LIN {X 0,Y 242.578,Z 857.441,A -85,B 0,C 180,E1 -19152.29,E2 -19152.29} C_VEL
LIN {X 0,Y 241.483,Z 861.061,A -85,B 0,C 180,E1 -19154.816,E2 -19154.816} C_VEL
LIN {X 0,Y 240.352,Z 864.916,A -85,B 0,C 180,E1 -19158.189,E2 -19158.189} C_VEL
LIN {X 0,Y 239.899,Z 867.777,A -85,B 0,C 180,E1 -19161.577,E2 -19161.577} C_VEL
LIN {X 0,Y 239.797,Z 869.672,A -85,B 0,C 180,E1 -19164.956,E2 -19164.956} C_VEL
LIN {X 0,Y 239.756,Z 870.35,A -85,B 0,C 180,E1 -19166.639,E2 -19166.639} C_VEL
LIN {X 0,Y 239.862,Z 870.828,A -85,B 0,C 180,E1 -19170,E2 -19170} C_VEL
LIN {X 0,Y 239.756,Z 870.35,A -85,B 0,C 180,E1 -19173.361,E2 -19173.361} C_VEL
LIN {X 0,Y 239.78,Z 868.917,A -85,B 0,C 180,E1 -19176.733,E2 -19176.733} C_VEL
LIN {X 0,Y 240.067,Z 866.522,A -85,B 0,C 180,E1 -19180.116,E2 -19180.116} C_VEL
LIN {X 0,Y 241.126,Z 862.101,A -85,B 0,C 180,E1 -19184.344,E2 -19184.344} C_VEL
LIN {X 0,Y 242.159,Z 858.729,A -85,B 0,C 180,E1 -19186.871,E2 -19186.871} C_VEL
LIN {X 0,Y 244.064,Z 853.224,A -85,B 0,C 180,E1 -19190.215,E2 -19190.215} C_VEL
LIN {X 0,Y 245.911,Z 848.361,A -85,B 0,C 180,E1 -19192.694,E2 -19192.694} C_VEL
LIN {X 0,Y 248.516,Z 841.742,A -85,B 0,C 180,E1 -19195.547,E2 -19195.547} C_VEL
LIN {X 0,Y 251.72,Z 834.036,A -85,B 0,C 180,E1 -19198.335,E2 -19198.335} C_VEL
LIN {X 0,Y 254.947,Z 826.486,A -85,B 0,C 180,E1 -19200.662,E2 -19200.662} C_VEL
LIN {X 0,Y 258.438,Z 817.9,A -85,B 0,C 180,E1 -19202.947,E2 -19202.947} C_VEL
LIN {X 0,Y 262.348,Z 808.111,A -85,B 0,C 180,E1 -19205.166,E2 -19205.166} C_VEL
LIN {X 0,Y 266.73,Z 796.887,A -85,B 0,C 180,E1 -19207.301,E2 -19207.301} C_VEL
LIN {X 0,Y 270.235,Z 787.33,A -85,B 0,C 180,E1 -19208.859,E2 -19208.859} C_VEL
LIN {X 0,Y 273.955,Z 776.523,A -85,B 0,C 180,E1 -19210.372,E2 -19210.372} C_VEL
LIN {X 0,Y 277.393,Z 765.586,A -85,B 0,C 180,E1 -19211.686,E2 -19211.686} C_VEL
LIN {X 0,Y 281.007,Z 752.933,A -85,B 0,C 180,E1 -19212.962,E2 -19212.962} C_VEL
LIN {X 0,Y 283.803,Z 741.946,A -85,B 0,C 180,E1 -19213.897,E2 -19213.897} C_VEL
LIN {X 0,Y 286.488,Z 729.861,A -85,B 0,C 180,E1 -19214.76,E2 -19214.76} C_VEL
LIN {X 0,Y 289.158,Z 715.743,A -85,B 0,C 180,E1 -19215.557,E2 -19215.557} C_VEL
LIN {X 0,Y 291.186,Z 702.376,A -85,B 0,C 180,E1 -19216.14,E2 -19216.14} C_VEL
LIN {X 0,Y 292.661,Z 688.923,A -85,B 0,C 180,E1 -19216.586,E2 -19216.586} C_VEL
LIN {X 0,Y 295.022,Z 651.638,A -85,B 0,C 180,E1 -19217.474,E2 -19217.474} C_VEL
LIN {X 0,Y 299.994,Z 567.021,A -85,B 0,C 180,E1 -19219.406,E2 -19219.406} C_VEL
LIN {X 0,Y 293.621,Z 552.933,A -85,B 0,C 180,E1 -19221.404,E2 -19221.404} C_VEL
LIN {X 0,Y 286.94,Z 539.628,A -85,B 0,C 180,E1 -19223.638,E2 -19223.638} C_VEL
LIN {X 0,Y 280.747,Z 528.524,A -85,B 0,C 180,E1 -19225.868,E2 -19225.868} C_VEL
LIN {X 0,Y 275.075,Z 519.016,A -85,B 0,C 180,E1 -19228.092,E2 -19228.092} C_VEL
LIN {X 0,Y 271.322,Z 513.261,A -85,B 0,C 180,E1 -19229.67,E2 -19229.67} C_VEL
LIN {X 0,Y 268.084,Z 508.973,A -85,B 0,C 180,E1 -19231.095,E2 -19231.095} C_VEL
LIN {X 0,Y 264.624,Z 504.496,A -85,B 0,C 180,E1 -19232.727,E2 -19232.727} C_VEL
LIN {X 0,Y 261.902,Z 501.009,A -85,B 0,C 180,E1 -19234.107,E2 -19234.107} C_VEL
LIN {X 0,Y 260.988,Z 499.86,A -85,B 0,C 180,E1 -19234.591,E2 -19234.591} C_VEL
LIN {X 0,Y 258.194,Z 496.863,A -85,B 0,C 180,E1 -19236.115,E2 -19236.115} C_VEL
LIN {X 0,Y 256.919,Z 494.86,A -85,B 0,C 180,E1 -19236.898,E2 -19236.898} C_VEL
LIN {X 0,Y 254.24,Z 492.546,A -85,B 0,C 180,E1 -19238.514,E2 -19238.514} C_VEL
LIN {X 0,Y 252.29,Z 489.301,A -85,B 0,C 180,E1 -19239.915,E2 -19239.915} C_VEL
LIN {X 0,Y 249.327,Z 487.104,A -85,B 0,C 180,E1 -19242.043,E2 -19242.043} C_VEL
LIN {X 0,Y 247.221,Z 483.628,A -85,B 0,C 180,E1 -19243.944,E2 -19243.944} C_VEL
LIN {X 0,Y 244.135,Z 481.605,A -85,B 0,C 180,E1 -19246.897,E2 -19246.897} C_VEL
LIN {X 0,Y 242.709,Z 479.452,A -85,B 0,C 180,E1 -19248.728,E2 -19248.728} C_VEL
LIN {X 0,Y 242.346,Z 478.039,A -85,B 0,C 180,E1 -19249.979,E2 -19249.979} C_VEL
LIN {X 0,Y 242.395,Z 477.56,A -85,B 0,C 180,E1 -19251.664,E2 -19251.664} C_VEL
LIN {X 0,Y 242.252,Z 477.542,A -85,B 0,C 180,E1 -19255.007,E2 -19255.007} C_VEL
LIN {X 0,Y 242.631,Z 477.502,A -85,B 0,C 180,E1 -19258.34,E2 -19258.34} C_VEL
LIN {X 0,Y 242.631,Z 477.483,A -85,B 0,C 180,E1 -19261.659,E2 -19261.659} C_VEL
LIN {X 0,Y 242.423,Z 477.508,A -85,B 0,C 180,E1 -19266.703,E2 -19266.703} C_VEL
LIN {X 0,Y 242.362,Z 477.788,A -85,B 0,C 180,E1 -19270.019,E2 -19270.019} C_VEL
LIN {X 0,Y 242.547,Z 478.94,A -85,B 0,C 180,E1 -19271.384,E2 -19271.384} C_VEL
LIN {X 0,Y 243.957,Z 481.47,A -85,B 0,C 180,E1 -19273.324,E2 -19273.324} C_VEL
LIN {X 0,Y 247.548,Z 484.008,A -85,B 0,C 180,E1 -19276.767,E2 -19276.767} C_VEL
LIN {X 0,Y 249.333,Z 487.146,A -85,B 0,C 180,E1 -19278.381,E2 -19278.381} C_VEL
LIN {X 0,Y 251.923,Z 489.174,A -85,B 0,C 180,E1 -19280.264,E2 -19280.264} C_VEL
LIN {X 0,Y 252.55,Z 489.767,A -85,B 0,C 180,E1 -19280.697,E2 -19280.697} C_VEL
LIN {X 0,Y 254.388,Z 492.805,A -85,B 0,C 180,E1 -19282.005,E2 -19282.005} C_VEL
LIN {X 0,Y 257.319,Z 495.333,A -85,B 0,C 180,E1 -19283.756,E2 -19283.756} C_VEL
LIN {X 0,Y 259.737,Z 498.727,A -85,B 0,C 180,E1 -19285.17,E2 -19285.17} C_VEL
LIN {X 0,Y 261.606,Z 500.6,A -85,B 0,C 180,E1 -19286.151,E2 -19286.151} C_VEL
LIN {X 0,Y 264.594,Z 504.494,A -85,B 0,C 180,E1 -19287.676,E2 -19287.676} C_VEL
LIN {X 0,Y 266.072,Z 506.379,A -85,B 0,C 180,E1 -19288.388,E2 -19288.388} C_VEL
LIN {X 0,Y 269.712,Z 511.008,A -85,B 0,C 180,E1 -19290.043,E2 -19290.043} C_VEL
LIN {X 0,Y 273.86,Z 516.542,A -85,B 0,C 180,E1 -19291.795,E2 -19291.795} C_VEL
LIN {X 0,Y 284.021,Z 529.623,A -85,B 0,C 180,E1 -19295.55,E2 -19295.55} C_VEL
LIN {X 0,Y 290.619,Z 536.586,A -85,B 0,C 180,E1 -19297.623,E2 -19297.623} C_VEL
LIN {X 0,Y 297.294,Z 542.946,A -85,B 0,C 180,E1 -19299.585,E2 -19299.585} C_VEL
LIN {X 0,Y 301.355,Z 546.585,A -85,B 0,C 180,E1 -19300.818,E2 -19300.818} C_VEL
LIN {X 0,Y 308.526,Z 553.049,A -85,B 0,C 180,E1 -19303.171,E2 -19303.171} C_VEL
LIN {X 0,Y 314.885,Z 558.94,A -85,B 0,C 180,E1 -19305.464,E2 -19305.464} C_VEL
LIN {X 0,Y 319.671,Z 563.42,A -85,B 0,C 180,E1 -19307.347,E2 -19307.347} C_VEL
LIN {X 0,Y 325.679,Z 569.287,A -85,B 0,C 180,E1 -19309.852,E2 -19309.852} C_VEL
LIN {X 0,Y 328.38,Z 571.697,A -85,B 0,C 180,E1 -19310.998,E2 -19310.998} C_VEL
LIN {X 0,Y 333.028,Z 576.13,A -85,B 0,C 180,E1 -19313.027,E2 -19313.027} C_VEL
LIN {X 0,Y 336.117,Z 578.85,A -85,B 0,C 180,E1 -19314.418,E2 -19314.418} C_VEL
LIN {X 0,Y 340.541,Z 582.947,A -85,B 0,C 180,E1 -19316.493,E2 -19316.493} C_VEL
LIN {X 0,Y 343.794,Z 585.63,A -85,B 0,C 180,E1 -19318.061,E2 -19318.061} C_VEL
LIN {X 0,Y 347.343,Z 589.012,A -85,B 0,C 180,E1 -19319.866,E2 -19319.866} C_VEL
LIN {X 0,Y 351.211,Z 592.136,A -85,B 0,C 180,E1 -19321.908,E2 -19321.908} C_VEL
LIN {X 0,Y 355.329,Z 596.17,A -85,B 0,C 180,E1 -19324.268,E2 -19324.268} C_VEL
LIN {X 0,Y 359.603,Z 599.246,A -85,B 0,C 180,E1 -19326.871,E2 -19326.871} C_VEL
LIN {X 0,Y 362.933,Z 602.606,A -85,B 0,C 180,E1 -19329.176,E2 -19329.176} C_VEL
LIN {X 0,Y 366.336,Z 605.042,A -85,B 0,C 180,E1 -19331.682,E2 -19331.682} C_VEL
LIN {X 0,Y 368.406,Z 606.343,A -85,B 0,C 180,E1 -19333.373,E2 -19333.373} C_VEL
LIN {X 0,Y 370.835,Z 609.08,A -85,B 0,C 180,E1 -19335.737,E2 -19335.737} C_VEL
LIN {X 0,Y 373.171,Z 611.039,A -85,B 0,C 180,E1 -19338.326,E2 -19338.326} C_VEL
LIN {X 0,Y 375.093,Z 612.069,A -85,B 0,C 180,E1 -19340.883,E2 -19340.883} C_VEL
LIN {X 0,Y 376.609,Z 612.81,A -85,B 0,C 180,E1 -19343.571,E2 -19343.571} C_VEL
LIN {X 0,Y 377.431,Z 613.376,A -85,B 0,C 180,E1 -19345.729,E2 -19345.729} C_VEL
LIN {X 0,Y 377.962,Z 613.558,A -85,B 0,C 180,E1 -19347.869,E2 -19347.869} C_VEL
LIN {X 0,Y 378.149,Z 613.625,A -85,B 0,C 180,E1 -19350,E2 -19350} C_VEL
LIN {X 0,Y 377.962,Z 613.559,A -85,B 0,C 180,E1 -19352.131,E2 -19352.131} C_VEL
LIN {X 0,Y 377.274,Z 613.269,A -85,B 0,C 180,E1 -19354.781,E2 -19354.781} C_VEL
LIN {X 0,Y 376.055,Z 612.562,A -85,B 0,C 180,E1 -19357.517,E2 -19357.517} C_VEL
LIN {X 0,Y 374.23,Z 611.679,A -85,B 0,C 180,E1 -19360.35,E2 -19360.35} C_VEL
LIN {X 0,Y 372.082,Z 610.203,A -85,B 0,C 180,E1 -19362.92,E2 -19362.92} C_VEL
LIN {X 0,Y 369.668,Z 607.864,A -85,B 0,C 180,E1 -19365.436,E2 -19365.436} C_VEL
LIN {X 0,Y 367.787,Z 605.761,A -85,B 0,C 180,E1 -19367.17,E2 -19367.17} C_VEL
LIN {X 0,Y 364.975,Z 604.141,A -85,B 0,C 180,E1 -19369.345,E2 -19369.345} C_VEL
LIN {X 0,Y 361.445,Z 601.277,A -85,B 0,C 180,E1 -19371.867,E2 -19371.867} C_VEL
LIN {X 0,Y 358.801,Z 598.546,A -85,B 0,C 180,E1 -19373.638,E2 -19373.638} C_VEL
LIN {X 0,Y 354.828,Z 595.742,A -85,B 0,C 180,E1 -19376.017,E2 -19376.017} C_VEL
LIN {X 0,Y 350.884,Z 591.778,A -85,B 0,C 180,E1 -19378.28,E2 -19378.28} C_VEL
LIN {X 0,Y 345.972,Z 587.873,A -85,B 0,C 180,E1 -19380.832,E2 -19380.832} C_VEL
LIN {X 0,Y 342.068,Z 584.093,A -85,B 0,C 180,E1 -19382.788,E2 -19382.788} C_VEL
LIN {X 0,Y 337.417,Z 580.192,A -85,B 0,C 180,E1 -19384.975,E2 -19384.975} C_VEL
LIN {X 0,Y 333.911,Z 576.796,A -85,B 0,C 180,E1 -19386.585,E2 -19386.585} C_VEL
LIN {X 0,Y 328.966,Z 572.338,A -85,B 0,C 180,E1 -19388.746,E2 -19388.746} C_VEL
LIN {X 0,Y 326.272,Z 569.703,A -85,B 0,C 180,E1 -19389.911,E2 -19389.911} C_VEL
LIN {X 0,Y 321.823,Z 565.579,A -85,B 0,C 180,E1 -19391.758,E2 -19391.758} C_VEL
LIN {X 0,Y 318.346,Z 562.26,A -85,B 0,C 180,E1 -19393.185,E2 -19393.185} C_VEL
LIN {X 0,Y 312.159,Z 556.385,A -85,B 0,C 180,E1 -19395.543,E2 -19395.543} C_VEL
LIN {X 0,Y 307.422,Z 551.98,A -85,B 0,C 180,E1 -19397.201,E2 -19397.201} C_VEL
LIN {X 0,Y 300.789,Z 546.044,A -85,B 0,C 180,E1 -19399.361,E2 -19399.361} C_VEL
LIN {X 0,Y 293.324,Z 539.281,A -85,B 0,C 180,E1 -19401.584,E2 -19401.584} C_VEL
LIN {X 0,Y 285.505,Z 531.293,A -85,B 0,C 180,E1 -19403.962,E2 -19403.962} C_VEL
LIN {X 0,Y 279.921,Z 524.607,A -85,B 0,C 180,E1 -19405.877,E2 -19405.877} C_VEL
LIN {X 0,Y 271.593,Z 513.467,A -85,B 0,C 180,E1 -19409.148,E2 -19409.148} C_VEL
LIN {X 0,Y 268.299,Z 509.207,A -85,B 0,C 180,E1 -19410.584,E2 -19410.584} C_VEL
LIN {X 0,Y 264.715,Z 504.61,A -85,B 0,C 180,E1 -19412.267,E2 -19412.267} C_VEL
LIN {X 0,Y 261.77,Z 500.861,A -85,B 0,C 180,E1 -19413.759,E2 -19413.759} C_VEL
LIN {X 0,Y 260.849,Z 499.688,A -85,B 0,C 180,E1 -19414.25,E2 -19414.25} C_VEL
LIN {X 0,Y 258.122,Z 496.718,A -85,B 0,C 180,E1 -19415.745,E2 -19415.745} C_VEL
LIN {X 0,Y 256.853,Z 494.821,A -85,B 0,C 180,E1 -19416.519,E2 -19416.519} C_VEL
LIN {X 0,Y 254.103,Z 492.457,A -85,B 0,C 180,E1 -19418.183,E2 -19418.183} C_VEL
LIN {X 0,Y 252.405,Z 489.438,A -85,B 0,C 180,E1 -19419.418,E2 -19419.418} C_VEL
LIN {X 0,Y 249.7,Z 487.548,A -85,B 0,C 180,E1 -19421.328,E2 -19421.328} C_VEL
LIN {X 0,Y 247.993,Z 484.981,A -85,B 0,C 180,E1 -19422.795,E2 -19422.795} C_VEL
LIN {X 0,Y 247.164,Z 483.61,A -85,B 0,C 180,E1 -19423.575,E2 -19423.575} C_VEL
LIN {X 0,Y 243.957,Z 481.47,A -85,B 0,C 180,E1 -19426.676,E2 -19426.676} C_VEL
LIN {X 0,Y 242.598,Z 479.136,A -85,B 0,C 180,E1 -19428.512,E2 -19428.512} C_VEL
LIN {X 0,Y 242.338,Z 478.057,A -85,B 0,C 180,E1 -19429.558,E2 -19429.558} C_VEL
LIN {X 0,Y 242.381,Z 477.587,A -85,B 0,C 180,E1 -19430.764,E2 -19430.764} C_VEL
LIN {X 0,Y 242.426,Z 477.509,A -85,B 0,C 180,E1 -19433.341,E2 -19433.341} C_VEL
LIN {X 0,Y 242.631,Z 477.485,A -85,B 0,C 180,E1 -19438.341,E2 -19438.341} C_VEL
LIN {X 0,Y 242.631,Z 477.504,A -85,B 0,C 180,E1 -19441.66,E2 -19441.66} C_VEL
LIN {X 0,Y 242.419,Z 477.527,A -85,B 0,C 180,E1 -19446.66,E2 -19446.66} C_VEL
LIN {X 0,Y 242.373,Z 477.818,A -85,B 0,C 180,E1 -19449.645,E2 -19449.645} C_VEL
LIN {X 0,Y 242.593,Z 479.137,A -85,B 0,C 180,E1 -19451.066,E2 -19451.066} C_VEL
LIN {X 0,Y 244.132,Z 481.628,A -85,B 0,C 180,E1 -19453.103,E2 -19453.103} C_VEL
LIN {X 0,Y 247.528,Z 483.951,A -85,B 0,C 180,E1 -19456.33,E2 -19456.33} C_VEL
LIN {X 0,Y 249.449,Z 487.231,A -85,B 0,C 180,E1 -19458.054,E2 -19458.054} C_VEL
LIN {X 0,Y 252.537,Z 489.602,A -85,B 0,C 180,E1 -19460.26,E2 -19460.26} C_VEL
LIN {X 0,Y 254.346,Z 492.684,A -85,B 0,C 180,E1 -19461.556,E2 -19461.556} C_VEL
LIN {X 0,Y 257.375,Z 495.471,A -85,B 0,C 180,E1 -19463.378,E2 -19463.378} C_VEL
LIN {X 0,Y 259.718,Z 498.74,A -85,B 0,C 180,E1 -19464.747,E2 -19464.747} C_VEL
LIN {X 0,Y 261.594,Z 500.527,A -85,B 0,C 180,E1 -19465.725,E2 -19465.725} C_VEL
LIN {X 0,Y 264.253,Z 504.142,A -85,B 0,C 180,E1 -19467.097,E2 -19467.097} C_VEL
LIN {X 0,Y 265.821,Z 505.972,A -85,B 0,C 180,E1 -19467.848,E2 -19467.848} C_VEL
LIN {X 0,Y 269.791,Z 511.206,A -85,B 0,C 180,E1 -19469.666,E2 -19469.666} C_VEL
LIN {X 0,Y 273.093,Z 515.902,A -85,B 0,C 180,E1 -19471.085,E2 -19471.085} C_VEL
LIN {X 0,Y 278.448,Z 524.496,A -85,B 0,C 180,E1 -19473.249,E2 -19473.249} C_VEL
LIN {X 0,Y 285.75,Z 537.328,A -85,B 0,C 180,E1 -19475.943,E2 -19475.943} C_VEL
LIN {X 0,Y 292.568,Z 550.783,A -85,B 0,C 180,E1 -19478.256,E2 -19478.256} C_VEL
LIN {X 0,Y 298.601,Z 563.806,A -85,B 0,C 180,E1 -19480.166,E2 -19480.166} C_VEL
LIN {X 0,Y 300.007,Z 567.051,A -85,B 0,C 180,E1 -19480.598,E2 -19480.598} C_VEL
LIN {X 0,Y 299.387,Z 577.69,A -85,B 0,C 180,E1 -19480.842,E2 -19480.842} C_VEL
LIN {X 0,Y 298.645,Z 583.54,A -85,B 0,C 180,E1 -19480.889,E2 -19480.889} C_VEL
LIN {X 0,Y 293.745,Z 602.654,A -85,B 0,C 180,E1 -19480.488,E2 -19480.488} C_VEL
LIN {X 0,Y 292.942,Z 608.51,A -85,B 0,C 180,E1 -19480.521,E2 -19480.521} C_VEL
LIN {X 0,Y 288.087,Z 685.999,A -85,B 0,C 180,E1 -19482.314,E2 -19482.314} C_VEL
LIN {X 0,Y 286.556,Z 700.167,A -85,B 0,C 180,E1 -19482.759,E2 -19482.759} C_VEL
LIN {X 0,Y 284.599,Z 713.234,A -85,B 0,C 180,E1 -19483.306,E2 -19483.306} C_VEL
LIN {X 0,Y 282.221,Z 725.93,A -85,B 0,C 180,E1 -19483.989,E2 -19483.989} C_VEL
LIN {X 0,Y 279.53,Z 738.313,A -85,B 0,C 180,E1 -19484.83,E2 -19484.83} C_VEL
LIN {X 0,Y 276.776,Z 749.24,A -85,B 0,C 180,E1 -19485.711,E2 -19485.711} C_VEL
LIN {X 0,Y 273.496,Z 760.877,A -85,B 0,C 180,E1 -19486.83,E2 -19486.83} C_VEL
LIN {X 0,Y 269.896,Z 772.398,A -85,B 0,C 180,E1 -19488.145,E2 -19488.145} C_VEL
LIN {X 0,Y 265.937,Z 783.688,A -85,B 0,C 180,E1 -19489.65,E2 -19489.65} C_VEL
LIN {X 0,Y 261.659,Z 795.329,A -85,B 0,C 180,E1 -19491.519,E2 -19491.519} C_VEL
LIN {X 0,Y 257.983,Z 804.349,A -85,B 0,C 180,E1 -19493.179,E2 -19493.179} C_VEL
LIN {X 0,Y 253.717,Z 814.554,A -85,B 0,C 180,E1 -19495.4,E2 -19495.4} C_VEL
LIN {X 0,Y 249.883,Z 823.512,A -85,B 0,C 180,E1 -19497.699,E2 -19497.699} C_VEL
LIN {X 0,Y 246.478,Z 831.405,A -85,B 0,C 180,E1 -19500.068,E2 -19500.068} C_VEL
LIN {X 0,Y 243.37,Z 838.369,A -85,B 0,C 180,E1 -19502.482,E2 -19502.482} C_VEL
LIN {X 0,Y 240.696,Z 844.59,A -85,B 0,C 180,E1 -19504.992,E2 -19504.992} C_VEL
LIN {X 0,Y 237.885,Z 851.464,A -85,B 0,C 180,E1 -19508.328,E2 -19508.328} C_VEL
LIN {X 0,Y 235.709,Z 857.228,A -85,B 0,C 180,E1 -19511.756,E2 -19511.756} C_VEL
LIN {X 0,Y 234.186,Z 861.889,A -85,B 0,C 180,E1 -19515.222,E2 -19515.222} C_VEL
LIN {X 0,Y 233.017,Z 866.311,A -85,B 0,C 180,E1 -19519.574,E2 -19519.574} C_VEL
LIN {X 0,Y 232.698,Z 868.707,A -85,B 0,C 180,E1 -19523.061,E2 -19523.061} C_VEL
LIN {X 0,Y 232.666,Z 870.14,A -85,B 0,C 180,E1 -19526.537,E2 -19526.537} C_VEL
LIN {X 0,Y 232.774,Z 870.619,A -85,B 0,C 180,E1 -19530,E2 -19530} C_VEL
LIN {X 0,Y 232.665,Z 870.14,A -85,B 0,C 180,E1 -19533.463,E2 -19533.463} C_VEL
LIN {X 0,Y 232.698,Z 868.706,A -85,B 0,C 180,E1 -19536.939,E2 -19536.939} C_VEL
LIN {X 0,Y 233.014,Z 866.311,A -85,B 0,C 180,E1 -19540.426,E2 -19540.426} C_VEL
LIN {X 0,Y 234.166,Z 861.888,A -85,B 0,C 180,E1 -19544.78,E2 -19544.78} C_VEL
LIN {X 0,Y 235.706,Z 857.227,A -85,B 0,C 180,E1 -19548.244,E2 -19548.244} C_VEL
LIN {X 0,Y 237.901,Z 851.464,A -85,B 0,C 180,E1 -19551.67,E2 -19551.67} C_VEL
LIN {X 0,Y 240.979,Z 843.955,A -85,B 0,C 180,E1 -19555.298,E2 -19555.298} C_VEL
LIN {X 0,Y 244.858,Z 835.031,A -85,B 0,C 180,E1 -19558.735,E2 -19558.735} C_VEL
LIN {X 0,Y 248.754,Z 826.272,A -85,B 0,C 180,E1 -19561.511,E2 -19561.511} C_VEL
LIN {X 0,Y 252.424,Z 817.687,A -85,B 0,C 180,E1 -19563.837,E2 -19563.837} C_VEL
LIN {X 0,Y 256.496,Z 807.898,A -85,B 0,C 180,E1 -19566.092,E2 -19566.092} C_VEL
LIN {X 0,Y 260.665,Z 797.681,A -85,B 0,C 180,E1 -19568.078,E2 -19568.078} C_VEL
LIN {X 0,Y 264.707,Z 787.119,A -85,B 0,C 180,E1 -19569.83,E2 -19569.83} C_VEL
LIN {X 0,Y 268.551,Z 776.312,A -85,B 0,C 180,E1 -19571.359,E2 -19571.359} C_VEL
LIN {X 0,Y 272.086,Z 765.375,A -85,B 0,C 180,E1 -19572.689,E2 -19572.689} C_VEL
LIN {X 0,Y 275.833,Z 752.723,A -85,B 0,C 180,E1 -19573.971,E2 -19573.971} C_VEL
LIN {X 0,Y 279.014,Z 740.52,A -85,B 0,C 180,E1 -19575.002,E2 -19575.002} C_VEL
LIN {X 0,Y 281.833,Z 728.015,A -85,B 0,C 180,E1 -19575.876,E2 -19575.876} C_VEL
LIN {X 0,Y 284.361,Z 714.767,A -85,B 0,C 180,E1 -19576.615,E2 -19576.615} C_VEL
LIN {X 0,Y 286.316,Z 702.167,A -85,B 0,C 180,E1 -19577.164,E2 -19577.164} C_VEL
LIN {X 0,Y 287.821,Z 688.713,A -85,B 0,C 180,E1 -19577.614,E2 -19577.614} C_VEL
LIN {X 0,Y 290.268,Z 651.428,A -85,B 0,C 180,E1 -19578.508,E2 -19578.508} C_VEL
LIN {X 0,Y 295.232,Z 570.658,A -85,B 0,C 180,E1 -19580.353,E2 -19580.353} C_VEL
LIN {X 0,Y 295.075,Z 569.346,A -85,B 0,C 180,E1 -19580.439,E2 -19580.439} C_VEL
LIN {X 0,Y 289.66,Z 557.204,A -85,B 0,C 180,E1 -19582.22,E2 -19582.22} C_VEL
LIN {X 0,Y 283.403,Z 544.435,A -85,B 0,C 180,E1 -19584.409,E2 -19584.409} C_VEL
LIN {X 0,Y 277.395,Z 533.505,A -85,B 0,C 180,E1 -19586.666,E2 -19586.666} C_VEL
LIN {X 0,Y 272.283,Z 524.699,A -85,B 0,C 180,E1 -19588.758,E2 -19588.758} C_VEL
LIN {X 0,Y 268.629,Z 519.018,A -85,B 0,C 180,E1 -19590.354,E2 -19590.354} C_VEL
LIN {X 0,Y 265.723,Z 515.06,A -85,B 0,C 180,E1 -19591.684,E2 -19591.684} C_VEL
LIN {X 0,Y 262.691,Z 511.029,A -85,B 0,C 180,E1 -19593.162,E2 -19593.162} C_VEL
LIN {X 0,Y 259.678,Z 507.134,A -85,B 0,C 180,E1 -19594.739,E2 -19594.739} C_VEL
LIN {X 0,Y 255.903,Z 502.701,A -85,B 0,C 180,E1 -19596.881,E2 -19596.881} C_VEL
LIN {X 0,Y 255.059,Z 501.423,A -85,B 0,C 180,E1 -19597.416,E2 -19597.416} C_VEL
LIN {X 0,Y 252.353,Z 498.873,A -85,B 0,C 180,E1 -19599.122,E2 -19599.122} C_VEL
LIN {X 0,Y 250.721,Z 496.044,A -85,B 0,C 180,E1 -19600.344,E2 -19600.344} C_VEL
LIN {X 0,Y 247.866,Z 493.803,A -85,B 0,C 180,E1 -19602.466,E2 -19602.466} C_VEL
LIN {X 0,Y 245.972,Z 490.48,A -85,B 0,C 180,E1 -19604.244,E2 -19604.244} C_VEL
LIN {X 0,Y 243.004,Z 488.542,A -85,B 0,C 180,E1 -19607.154,E2 -19607.154} C_VEL
LIN {X 0,Y 241.462,Z 486.137,A -85,B 0,C 180,E1 -19609.2,E2 -19609.2} C_VEL
LIN {X 0,Y 240.567,Z 484.589,A -85,B 0,C 180,E1 -19610.625,E2 -19610.625} C_VEL
LIN {X 0,Y 237.598,Z 482.494,A -85,B 0,C 180,E1 -19618.305,E2 -19618.305} C_VEL
LIN {X 0,Y 237.552,Z 482.451,A -85,B 0,C 180,E1 -19621.695,E2 -19621.695} C_VEL
LIN {X 0,Y 240.611,Z 484.615,A -85,B 0,C 180,E1 -19629.858,E2 -19629.858} C_VEL
LIN {X 0,Y 241.398,Z 486.024,A -85,B 0,C 180,E1 -19631.12,E2 -19631.12} C_VEL
LIN {X 0,Y 243.095,Z 488.685,A -85,B 0,C 180,E1 -19633.372,E2 -19633.372} C_VEL
LIN {X 0,Y 246.11,Z 490.714,A -85,B 0,C 180,E1 -19636.308,E2 -19636.308} C_VEL
LIN {X 0,Y 247.758,Z 493.692,A -85,B 0,C 180,E1 -19637.861,E2 -19637.861} C_VEL
LIN {X 0,Y 250.398,Z 495.956,A -85,B 0,C 180,E1 -19639.859,E2 -19639.859} C_VEL
LIN {X 0,Y 251.045,Z 496.8,A -85,B 0,C 180,E1 -19640.338,E2 -19640.338} C_VEL
LIN {X 0,Y 253.246,Z 499.978,A -85,B 0,C 180,E1 -19641.895,E2 -19641.895} C_VEL
LIN {X 0,Y 255.524,Z 502.015,A -85,B 0,C 180,E1 -19643.289,E2 -19643.289} C_VEL
LIN {X 0,Y 258.351,Z 505.71,A -85,B 0,C 180,E1 -19644.96,E2 -19644.96} C_VEL
LIN {X 0,Y 259.726,Z 507.27,A -85,B 0,C 180,E1 -19645.708,E2 -19645.708} C_VEL
LIN {X 0,Y 262.821,Z 511.168,A -85,B 0,C 180,E1 -19647.318,E2 -19647.318} C_VEL
LIN {X 0,Y 267.62,Z 517.578,A -85,B 0,C 180,E1 -19649.606,E2 -19649.606} C_VEL
LIN {X 0,Y 270.907,Z 522.015,A -85,B 0,C 180,E1 -19651.043,E2 -19651.043} C_VEL
LIN {X 0,Y 281.495,Z 535.867,A -85,B 0,C 180,E1 -19655.092,E2 -19655.092} C_VEL
LIN {X 0,Y 287.919,Z 542.744,A -85,B 0,C 180,E1 -19657.166,E2 -19657.166} C_VEL
LIN {X 0,Y 295.192,Z 549.568,A -85,B 0,C 180,E1 -19659.295,E2 -19659.295} C_VEL
LIN {X 0,Y 302.425,Z 556.061,A -85,B 0,C 180,E1 -19661.525,E2 -19661.525} C_VEL
LIN {X 0,Y 305.86,Z 559.068,A -85,B 0,C 180,E1 -19662.644,E2 -19662.644} C_VEL
LIN {X 0,Y 310.698,Z 563.406,A -85,B 0,C 180,E1 -19664.317,E2 -19664.317} C_VEL
LIN {X 0,Y 316.854,Z 569.239,A -85,B 0,C 180,E1 -19666.633,E2 -19666.633} C_VEL
LIN {X 0,Y 319.938,Z 572.14,A -85,B 0,C 180,E1 -19667.879,E2 -19667.879} C_VEL
LIN {X 0,Y 324.807,Z 576.641,A -85,B 0,C 180,E1 -19669.898,E2 -19669.898} C_VEL
LIN {X 0,Y 331.048,Z 582.552,A -85,B 0,C 180,E1 -19672.593,E2 -19672.593} C_VEL
LIN {X 0,Y 334.327,Z 585.361,A -85,B 0,C 180,E1 -19674.047,E2 -19674.047} C_VEL
LIN {X 0,Y 338.74,Z 589.487,A -85,B 0,C 180,E1 -19676.087,E2 -19676.087} C_VEL
LIN {X 0,Y 342.282,Z 592.37,A -85,B 0,C 180,E1 -19677.779,E2 -19677.779} C_VEL
LIN {X 0,Y 345.934,Z 595.822,A -85,B 0,C 180,E1 -19679.627,E2 -19679.627} C_VEL
LIN {X 0,Y 349.861,Z 598.969,A -85,B 0,C 180,E1 -19681.672,E2 -19681.672} C_VEL
LIN {X 0,Y 353.995,Z 602.979,A -85,B 0,C 180,E1 -19684.034,E2 -19684.034} C_VEL
LIN {X 0,Y 358.415,Z 606.21,A -85,B 0,C 180,E1 -19686.701,E2 -19686.701} C_VEL
LIN {X 0,Y 361.742,Z 609.481,A -85,B 0,C 180,E1 -19688.965,E2 -19688.965} C_VEL
LIN {X 0,Y 365.198,Z 611.969,A -85,B 0,C 180,E1 -19691.481,E2 -19691.481} C_VEL
LIN {X 0,Y 367.292,Z 613.234,A -85,B 0,C 180,E1 -19693.172,E2 -19693.172} C_VEL
LIN {X 0,Y 369.659,Z 615.916,A -85,B 0,C 180,E1 -19695.443,E2 -19695.443} C_VEL
LIN {X 0,Y 372.051,Z 617.909,A -85,B 0,C 180,E1 -19698.008,E2 -19698.008} C_VEL
LIN {X 0,Y 374.024,Z 619.031,A -85,B 0,C 180,E1 -19700.607,E2 -19700.607} C_VEL
LIN {X 0,Y 375.395,Z 619.698,A -85,B 0,C 180,E1 -19702.855,E2 -19702.855} C_VEL
LIN {X 0,Y 376.404,Z 620.322,A -85,B 0,C 180,E1 -19705.208,E2 -19705.208} C_VEL
LIN {X 0,Y 377.097,Z 620.604,A -85,B 0,C 180,E1 -19707.864,E2 -19707.864} C_VEL
LIN {X 0,Y 377.284,Z 620.671,A -85,B 0,C 180,E1 -19710,E2 -19710} C_VEL
LIN {X 0,Y 377.097,Z 620.604,A -85,B 0,C 180,E1 -19712.136,E2 -19712.136} C_VEL
LIN {X 0,Y 376.404,Z 620.315,A -85,B 0,C 180,E1 -19714.793,E2 -19714.793} C_VEL
LIN {X 0,Y 375.174,Z 619.606,A -85,B 0,C 180,E1 -19717.535,E2 -19717.535} C_VEL
LIN {X 0,Y 373.344,Z 618.716,A -85,B 0,C 180,E1 -19720.375,E2 -19720.375} C_VEL
LIN {X 0,Y 371.178,Z 617.229,A -85,B 0,C 180,E1 -19722.952,E2 -19722.952} C_VEL
LIN {X 0,Y 368.74,Z 614.945,A -85,B 0,C 180,E1 -19725.476,E2 -19725.476} C_VEL
LIN {X 0,Y 366.978,Z 612.865,A -85,B 0,C 180,E1 -19727.109,E2 -19727.109} C_VEL
LIN {X 0,Y 364.011,Z 611.208,A -85,B 0,C 180,E1 -19729.396,E2 -19729.396} C_VEL
LIN {X 0,Y 360.329,Z 608.252,A -85,B 0,C 180,E1 -19732.005,E2 -19732.005} C_VEL
LIN {X 0,Y 357.56,Z 605.426,A -85,B 0,C 180,E1 -19733.848,E2 -19733.848} C_VEL
LIN {X 0,Y 353.634,Z 602.681,A -85,B 0,C 180,E1 -19736.174,E2 -19736.174} C_VEL
LIN {X 0,Y 349.592,Z 598.655,A -85,B 0,C 180,E1 -19738.48,E2 -19738.48} C_VEL
LIN {X 0,Y 344.431,Z 594.52,A -85,B 0,C 180,E1 -19741.147,E2 -19741.147} C_VEL
LIN {X 0,Y 340.545,Z 590.849,A -85,B 0,C 180,E1 -19743.056,E2 -19743.056} C_VEL
LIN {X 0,Y 335.681,Z 586.75,A -85,B 0,C 180,E1 -19745.332,E2 -19745.332} C_VEL
LIN {X 0,Y 332.197,Z 583.426,A -85,B 0,C 180,E1 -19746.914,E2 -19746.914} C_VEL
LIN {X 0,Y 327.107,Z 578.852,A -85,B 0,C 180,E1 -19749.121,E2 -19749.121} C_VEL
LIN {X 0,Y 324.594,Z 576.41,A -85,B 0,C 180,E1 -19750.192,E2 -19750.192} C_VEL
LIN {X 0,Y 320.057,Z 572.252,A -85,B 0,C 180,E1 -19752.072,E2 -19752.072} C_VEL
LIN {X 0,Y 316.857,Z 569.206,A -85,B 0,C 180,E1 -19753.368,E2 -19753.368} C_VEL
LIN {X 0,Y 311.828,Z 564.352,A -85,B 0,C 180,E1 -19755.287,E2 -19755.287} C_VEL
LIN {X 0,Y 306.361,Z 559.567,A -85,B 0,C 180,E1 -19757.184,E2 -19757.184} C_VEL
LIN {X 0,Y 302.676,Z 556.242,A -85,B 0,C 180,E1 -19758.397,E2 -19758.397} C_VEL
LIN {X 0,Y 297.62,Z 551.673,A -85,B 0,C 180,E1 -19759.97,E2 -19759.97} C_VEL
LIN {X 0,Y 290.602,Z 545.429,A -85,B 0,C 180,E1 -19762.03,E2 -19762.03} C_VEL
LIN {X 0,Y 282.646,Z 537.176,A -85,B 0,C 180,E1 -19764.518,E2 -19764.518} C_VEL
LIN {X 0,Y 277.149,Z 530.482,A -85,B 0,C 180,E1 -19766.466,E2 -19766.466} C_VEL
LIN {X 0,Y 269.11,Z 519.565,A -85,B 0,C 180,E1 -19769.732,E2 -19769.732} C_VEL
LIN {X 0,Y 265.849,Z 515.227,A -85,B 0,C 180,E1 -19771.209,E2 -19771.209} C_VEL
LIN {X 0,Y 262.353,Z 510.71,A -85,B 0,C 180,E1 -19772.91,E2 -19772.91} C_VEL
LIN {X 0,Y 258.77,Z 506.065,A -85,B 0,C 180,E1 -19774.817,E2 -19774.817} C_VEL
LIN {X 0,Y 255.96,Z 502.753,A -85,B 0,C 180,E1 -19776.432,E2 -19776.432} C_VEL
LIN {X 0,Y 254.918,Z 501.331,A -85,B 0,C 180,E1 -19777.082,E2 -19777.082} C_VEL
LIN {X 0,Y 252.128,Z 498.64,A -85,B 0,C 180,E1 -19778.857,E2 -19778.857} C_VEL
LIN {X 0,Y 250.629,Z 496.115,A -85,B 0,C 180,E1 -19779.98,E2 -19779.98} C_VEL
LIN {X 0,Y 247.872,Z 493.859,A -85,B 0,C 180,E1 -19782.041,E2 -19782.041} C_VEL
LIN {X 0,Y 246.151,Z 490.824,A -85,B 0,C 180,E1 -19783.648,E2 -19783.648} C_VEL
LIN {X 0,Y 242.499,Z 487.971,A -85,B 0,C 180,E1 -19787.34,E2 -19787.34} C_VEL
LIN {X 0,Y 240.749,Z 484.834,A -85,B 0,C 180,E1 -19789.913,E2 -19789.913} C_VEL
LIN {X 0,Y 238.882,Z 483.667,A -85,B 0,C 180,E1 -19793.242,E2 -19793.242} C_VEL
LIN {X 0,Y 237.554,Z 482.432,A -85,B 0,C 180,E1 -19798.305,E2 -19798.305} C_VEL
LIN {X 0,Y 237.644,Z 482.643,A -85,B 0,C 180,E1 -19802.119,E2 -19802.119} C_VEL
LIN {X 0,Y 240.562,Z 484.6,A -85,B 0,C 180,E1 -19809.37,E2 -19809.37} C_VEL
LIN {X 0,Y 241.46,Z 486.151,A -85,B 0,C 180,E1 -19810.8,E2 -19810.8} C_VEL
LIN {X 0,Y 243.091,Z 488.651,A -85,B 0,C 180,E1 -19812.948,E2 -19812.948} C_VEL
LIN {X 0,Y 246.219,Z 490.88,A -85,B 0,C 180,E1 -19815.997,E2 -19815.997} C_VEL
LIN {X 0,Y 247.867,Z 493.798,A -85,B 0,C 180,E1 -19817.534,E2 -19817.534} C_VEL
LIN {X 0,Y 250.909,Z 496.406,A -85,B 0,C 180,E1 -19819.805,E2 -19819.805} C_VEL
LIN {X 0,Y 253.09,Z 499.777,A -85,B 0,C 180,E1 -19821.375,E2 -19821.375} C_VEL
LIN {X 0,Y 255.505,Z 502.014,A -85,B 0,C 180,E1 -19822.863,E2 -19822.863} C_VEL
LIN {X 0,Y 258.255,Z 505.647,A -85,B 0,C 180,E1 -19824.494,E2 -19824.494} C_VEL
LIN {X 0,Y 259.759,Z 507.304,A -85,B 0,C 180,E1 -19825.31,E2 -19825.31} C_VEL
LIN {X 0,Y 262.873,Z 511.192,A -85,B 0,C 180,E1 -19826.926,E2 -19826.926} C_VEL
LIN {X 0,Y 267.586,Z 517.608,A -85,B 0,C 180,E1 -19829.179,E2 -19829.179} C_VEL
LIN {X 0,Y 270.501,Z 521.857,A -85,B 0,C 180,E1 -19830.474,E2 -19830.474} C_VEL
LIN {X 0,Y 275.882,Z 530.82,A -85,B 0,C 180,E1 -19832.731,E2 -19832.731} C_VEL
LIN {X 0,Y 282.246,Z 542.147,A -85,B 0,C 180,E1 -19835.166,E2 -19835.166} C_VEL
LIN {X 0,Y 289.088,Z 556.038,A -85,B 0,C 180,E1 -19837.588,E2 -19837.588} C_VEL
LIN {X 0,Y 294.539,Z 568.037,A -85,B 0,C 180,E1 -19839.387,E2 -19839.387} C_VEL
LIN {X 0,Y 295.202,Z 569.643,A -85,B 0,C 180,E1 -19839.602,E2 -19839.602} C_VEL
LIN {X 0,Y 292.942,Z 608.51,A -85,B 0,C 180,E1 -19840.521,E2 -19840.521} C_VEL
LIN {X 0,Y 292.136,Z 614.368,A -85,B 0,C 180,E1 -19840.553,E2 -19840.553} C_VEL
LIN {X 0,Y 287.172,Z 633.471,A -85,B 0,C 180,E1 -19840.119,E2 -19840.119} C_VEL
LIN {X 0,Y 286.372,Z 639.328,A -85,B 0,C 180,E1 -19840.153,E2 -19840.153} C_VEL
LIN {X 0,Y 283.213,Z 687.144,A -85,B 0,C 180,E1 -19841.287,E2 -19841.287} C_VEL
LIN {X 0,Y 281.653,Z 700.957,A -85,B 0,C 180,E1 -19841.736,E2 -19841.736} C_VEL
LIN {X 0,Y 279.637,Z 713.79,A -85,B 0,C 180,E1 -19842.284,E2 -19842.284} C_VEL
LIN {X 0,Y 277.285,Z 725.873,A -85,B 0,C 180,E1 -19842.939,E2 -19842.939} C_VEL
LIN {X 0,Y 274.599,Z 737.857,A -85,B 0,C 180,E1 -19843.753,E2 -19843.753} C_VEL
LIN {X 0,Y 271.698,Z 749.029,A -85,B 0,C 180,E1 -19844.657,E2 -19844.657} C_VEL
LIN {X 0,Y 268.313,Z 760.665,A -85,B 0,C 180,E1 -19845.783,E2 -19845.783} C_VEL
LIN {X 0,Y 264.149,Z 773.491,A -85,B 0,C 180,E1 -19847.278,E2 -19847.278} C_VEL
LIN {X 0,Y 260.084,Z 784.62,A -85,B 0,C 180,E1 -19848.803,E2 -19848.803} C_VEL
LIN {X 0,Y 256.458,Z 794.126,A -85,B 0,C 180,E1 -19850.339,E2 -19850.339} C_VEL
LIN {X 0,Y 252.256,Z 804.136,A -85,B 0,C 180,E1 -19852.199,E2 -19852.199} C_VEL
LIN {X 0,Y 247.838,Z 814.342,A -85,B 0,C 180,E1 -19854.457,E2 -19854.457} C_VEL
LIN {X 0,Y 243.81,Z 823.299,A -85,B 0,C 180,E1 -19856.792,E2 -19856.792} C_VEL
LIN {X 0,Y 240.253,Z 831.192,A -85,B 0,C 180,E1 -19859.209,E2 -19859.209} C_VEL
LIN {X 0,Y 236.994,Z 838.155,A -85,B 0,C 180,E1 -19861.675,E2 -19861.675} C_VEL
LIN {X 0,Y 234.249,Z 844.21,A -85,B 0,C 180,E1 -19864.167,E2 -19864.167} C_VEL
LIN {X 0,Y 231.207,Z 851.251,A -85,B 0,C 180,E1 -19867.669,E2 -19867.669} C_VEL
LIN {X 0,Y 228.878,Z 857.015,A -85,B 0,C 180,E1 -19871.191,E2 -19871.191} C_VEL
LIN {X 0,Y 227.627,Z 860.635,A -85,B 0,C 180,E1 -19873.867,E2 -19873.867} C_VEL
LIN {X 0,Y 226.331,Z 864.492,A -85,B 0,C 180,E1 -19877.446,E2 -19877.446} C_VEL
LIN {X 0,Y 225.752,Z 867.354,A -85,B 0,C 180,E1 -19881.045,E2 -19881.045} C_VEL
LIN {X 0,Y 225.587,Z 869.25,A -85,B 0,C 180,E1 -19884.637,E2 -19884.637} C_VEL
LIN {X 0,Y 225.58,Z 869.93,A -85,B 0,C 180,E1 -19886.428,E2 -19886.428} C_VEL
LIN {X 0,Y 225.688,Z 870.409,A -85,B 0,C 180,E1 -19890,E2 -19890} C_VEL
LIN {X 0,Y 225.579,Z 869.93,A -85,B 0,C 180,E1 -19893.572,E2 -19893.572} C_VEL
LIN {X 0,Y 225.607,Z 868.495,A -85,B 0,C 180,E1 -19897.158,E2 -19897.158} C_VEL
LIN {X 0,Y 225.979,Z 866.099,A -85,B 0,C 180,E1 -19900.754,E2 -19900.754} C_VEL
LIN {X 0,Y 227.23,Z 861.676,A -85,B 0,C 180,E1 -19905.242,E2 -19905.242} C_VEL
LIN {X 0,Y 228.396,Z 858.303,A -85,B 0,C 180,E1 -19907.921,E2 -19907.921} C_VEL
LIN {X 0,Y 230.545,Z 852.796,A -85,B 0,C 180,E1 -19911.457,E2 -19911.457} C_VEL
LIN {X 0,Y 232.642,Z 847.934,A -85,B 0,C 180,E1 -19914.068,E2 -19914.068} C_VEL
LIN {X 0,Y 236,Z 840.261,A -85,B 0,C 180,E1 -19917.489,E2 -19917.489} C_VEL
LIN {X 0,Y 239.116,Z 833.609,A -85,B 0,C 180,E1 -19919.977,E2 -19919.977} C_VEL
LIN {X 0,Y 242.626,Z 826.059,A -85,B 0,C 180,E1 -19922.403,E2 -19922.403} C_VEL
LIN {X 0,Y 246.445,Z 817.473,A -85,B 0,C 180,E1 -19924.774,E2 -19924.774} C_VEL
LIN {X 0,Y 250.734,Z 807.686,A -85,B 0,C 180,E1 -19927.058,E2 -19927.058} C_VEL
LIN {X 0,Y 255.053,Z 797.469,A -85,B 0,C 180,E1 -19929.073,E2 -19929.073} C_VEL
LIN {X 0,Y 259.235,Z 786.907,A -85,B 0,C 180,E1 -19930.846,E2 -19930.846} C_VEL
LIN {X 0,Y 263.195,Z 776.099,A -85,B 0,C 180,E1 -19932.394,E2 -19932.394} C_VEL
LIN {X 0,Y 266.879,Z 765.164,A -85,B 0,C 180,E1 -19933.729,E2 -19933.729} C_VEL
LIN {X 0,Y 270.247,Z 754.253,A -85,B 0,C 180,E1 -19934.861,E2 -19934.861} C_VEL
LIN {X 0,Y 273.714,Z 741.525,A -85,B 0,C 180,E1 -19935.966,E2 -19935.966} C_VEL
LIN {X 0,Y 276.623,Z 729.258,A -85,B 0,C 180,E1 -19936.843,E2 -19936.843} C_VEL
LIN {X 0,Y 279.388,Z 715.323,A -85,B 0,C 180,E1 -19937.639,E2 -19937.639} C_VEL
LIN {X 0,Y 281.541,Z 701.957,A -85,B 0,C 180,E1 -19938.223,E2 -19938.223} C_VEL
LIN {X 0,Y 283.088,Z 688.504,A -85,B 0,C 180,E1 -19938.675,E2 -19938.675} C_VEL
LIN {X 0,Y 285.618,Z 651.219,A -85,B 0,C 180,E1 -19939.574,E2 -19939.574} C_VEL
LIN {X 0,Y 290.593,Z 572.371,A -85,B 0,C 180,E1 -19941.396,E2 -19941.396} C_VEL
LIN {X 0,Y 284.57,Z 558.845,A -85,B 0,C 180,E1 -19943.484,E2 -19943.484} C_VEL
LIN {X 0,Y 278.81,Z 547.184,A -85,B 0,C 180,E1 -19945.617,E2 -19945.617} C_VEL
LIN {X 0,Y 272.143,Z 534.849,A -85,B 0,C 180,E1 -19948.307,E2 -19948.307} C_VEL
LIN {X 0,Y 266.427,Z 525.4,A -85,B 0,C 180,E1 -19950.844,E2 -19950.844} C_VEL
LIN {X 0,Y 263.105,Z 520.843,A -85,B 0,C 180,E1 -19952.417,E2 -19952.417} C_VEL
LIN {X 0,Y 260.082,Z 516.841,A -85,B 0,C 180,E1 -19953.953,E2 -19953.953} C_VEL
LIN {X 0,Y 256.954,Z 512.671,A -85,B 0,C 180,E1 -19955.677,E2 -19955.677} C_VEL
LIN {X 0,Y 254.016,Z 509.117,A -85,B 0,C 180,E1 -19957.425,E2 -19957.425} C_VEL
LIN {X 0,Y 253.14,Z 507.95,A -85,B 0,C 180,E1 -19957.988,E2 -19957.988} C_VEL
LIN {X 0,Y 250.31,Z 504.907,A -85,B 0,C 180,E1 -19959.876,E2 -19959.876} C_VEL
LIN {X 0,Y 249.06,Z 502.744,A -85,B 0,C 180,E1 -19960.85,E2 -19960.85} C_VEL
LIN {X 0,Y 246.195,Z 500.203,A -85,B 0,C 180,E1 -19963.093,E2 -19963.093} C_VEL
LIN {X 0,Y 244.677,Z 497.361,A -85,B 0,C 180,E1 -19964.589,E2 -19964.589} C_VEL
LIN {X 0,Y 241.879,Z 495.476,A -85,B 0,C 180,E1 -19967.413,E2 -19967.413} C_VEL
LIN {X 0,Y 240.305,Z 492.985,A -85,B 0,C 180,E1 -19969.574,E2 -19969.574} C_VEL
LIN {X 0,Y 239.557,Z 491.568,A -85,B 0,C 180,E1 -19970.826,E2 -19970.826} C_VEL
LIN {X 0,Y 236.733,Z 489.544,A -85,B 0,C 180,E1 -19978.298,E2 -19978.298} C_VEL
LIN {X 0,Y 236.686,Z 489.504,A -85,B 0,C 180,E1 -19981.701,E2 -19981.701} C_VEL
LIN {X 0,Y 239.603,Z 491.609,A -85,B 0,C 180,E1 -19989.664,E2 -19989.664} C_VEL
LIN {X 0,Y 240.307,Z 493.035,A -85,B 0,C 180,E1 -19990.851,E2 -19990.851} C_VEL
LIN {X 0,Y 242.058,Z 495.697,A -85,B 0,C 180,E1 -19993.217,E2 -19993.217} C_VEL
LIN {X 0,Y 244.727,Z 497.566,A -85,B 0,C 180,E1 -19995.891,E2 -19995.891} C_VEL
LIN {X 0,Y 246.514,Z 500.655,A -85,B 0,C 180,E1 -19997.605,E2 -19997.605} C_VEL
LIN {X 0,Y 249.309,Z 503.263,A -85,B 0,C 180,E1 -19999.772,E2 -19999.772} C_VEL
LIN {X 0,Y 251.69,Z 506.693,A -85,B 0,C 180,E1 -20001.509,E2 -20001.509} C_VEL
LIN {X 0,Y 253.827,Z 508.728,A -85,B 0,C 180,E1 -20002.861,E2 -20002.861} C_VEL
LIN {X 0,Y 256.633,Z 512.36,A -85,B 0,C 180,E1 -20004.56,E2 -20004.56} C_VEL
LIN {X 0,Y 257.798,Z 513.798,A -85,B 0,C 180,E1 -20005.219,E2 -20005.219} C_VEL
LIN {X 0,Y 261.937,Z 519.277,A -85,B 0,C 180,E1 -20007.418,E2 -20007.418} C_VEL
LIN {X 0,Y 265.189,Z 523.595,A -85,B 0,C 180,E1 -20008.993,E2 -20008.993} C_VEL
LIN {X 0,Y 270.62,Z 531.107,A -85,B 0,C 180,E1 -20011.4,E2 -20011.4} C_VEL
LIN {X 0,Y 278.672,Z 541.789,A -85,B 0,C 180,E1 -20014.517,E2 -20014.517} C_VEL
LIN {X 0,Y 285.218,Z 548.859,A -85,B 0,C 180,E1 -20016.693,E2 -20016.693} C_VEL
LIN {X 0,Y 292.627,Z 555.878,A -85,B 0,C 180,E1 -20018.897,E2 -20018.897} C_VEL
LIN {X 0,Y 300.391,Z 562.684,A -85,B 0,C 180,E1 -20021.233,E2 -20021.233} C_VEL
LIN {X 0,Y 305.891,Z 567.628,A -85,B 0,C 180,E1 -20023.029,E2 -20023.029} C_VEL
LIN {X 0,Y 311.725,Z 572.81,A -85,B 0,C 180,E1 -20025.061,E2 -20025.061} C_VEL
LIN {X 0,Y 318.046,Z 578.68,A -85,B 0,C 180,E1 -20027.515,E2 -20027.515} C_VEL
LIN {X 0,Y 323.205,Z 583.407,A -85,B 0,C 180,E1 -20029.645,E2 -20029.645} C_VEL
LIN {X 0,Y 329.404,Z 589.249,A -85,B 0,C 180,E1 -20032.3,E2 -20032.3} C_VEL
LIN {X 0,Y 332.882,Z 592.255,A -85,B 0,C 180,E1 -20033.832,E2 -20033.832} C_VEL
LIN {X 0,Y 337.436,Z 596.41,A -85,B 0,C 180,E1 -20035.93,E2 -20035.93} C_VEL
LIN {X 0,Y 340.969,Z 599.306,A -85,B 0,C 180,E1 -20037.595,E2 -20037.595} C_VEL
LIN {X 0,Y 345.059,Z 603.048,A -85,B 0,C 180,E1 -20039.658,E2 -20039.658} C_VEL
LIN {X 0,Y 348.615,Z 605.893,A -85,B 0,C 180,E1 -20041.504,E2 -20041.504} C_VEL
LIN {X 0,Y 352.789,Z 609.91,A -85,B 0,C 180,E1 -20043.87,E2 -20043.87} C_VEL
LIN {X 0,Y 357.077,Z 612.965,A -85,B 0,C 180,E1 -20046.429,E2 -20046.429} C_VEL
LIN {X 0,Y 360.543,Z 616.341,A -85,B 0,C 180,E1 -20048.742,E2 -20048.742} C_VEL
LIN {X 0,Y 364.02,Z 618.871,A -85,B 0,C 180,E1 -20051.276,E2 -20051.276} C_VEL
LIN {X 0,Y 366.385,Z 620.358,A -85,B 0,C 180,E1 -20053.158,E2 -20053.158} C_VEL
LIN {X 0,Y 368.795,Z 623.01,A -85,B 0,C 180,E1 -20055.462,E2 -20055.462} C_VEL
LIN {X 0,Y 371.145,Z 624.958,A -85,B 0,C 180,E1 -20057.978,E2 -20057.978} C_VEL
LIN {X 0,Y 372.902,Z 625.954,A -85,B 0,C 180,E1 -20060.234,E2 -20060.234} C_VEL
LIN {X 0,Y 374.532,Z 626.749,A -85,B 0,C 180,E1 -20062.864,E2 -20062.864} C_VEL
LIN {X 0,Y 375.534,Z 627.368,A -85,B 0,C 180,E1 -20065.197,E2 -20065.197} C_VEL
LIN {X 0,Y 376.232,Z 627.636,A -85,B 0,C 180,E1 -20067.859,E2 -20067.859} C_VEL
LIN {X 0,Y 376.418,Z 627.717,A -85,B 0,C 180,E1 -20070,E2 -20070} C_VEL
LIN {X 0,Y 376.232,Z 627.636,A -85,B 0,C 180,E1 -20072.141,E2 -20072.141} C_VEL
LIN {X 0,Y 375.535,Z 627.361,A -85,B 0,C 180,E1 -20074.804,E2 -20074.804} C_VEL
LIN {X 0,Y 374.296,Z 626.626,A -85,B 0,C 180,E1 -20077.552,E2 -20077.552} C_VEL
LIN {X 0,Y 372.456,Z 625.743,A -85,B 0,C 180,E1 -20080.4,E2 -20080.4} C_VEL
LIN {X 0,Y 370.271,Z 624.283,A -85,B 0,C 180,E1 -20082.984,E2 -20082.984} C_VEL
LIN {X 0,Y 367.901,Z 622.085,A -85,B 0,C 180,E1 -20085.432,E2 -20085.432} C_VEL
LIN {X 0,Y 365.824,Z 619.806,A -85,B 0,C 180,E1 -20087.314,E2 -20087.314} C_VEL
LIN {X 0,Y 362.85,Z 618.099,A -85,B 0,C 180,E1 -20089.601,E2 -20089.601} C_VEL
LIN {X 0,Y 359.109,Z 615.119,A -85,B 0,C 180,E1 -20092.216,E2 -20092.216} C_VEL
LIN {X 0,Y 356.327,Z 612.31,A -85,B 0,C 180,E1 -20094.058,E2 -20094.058} C_VEL
LIN {X 0,Y 352.453,Z 609.617,A -85,B 0,C 180,E1 -20096.324,E2 -20096.324} C_VEL
LIN {X 0,Y 348.36,Z 605.669,A -85,B 0,C 180,E1 -20098.63,E2 -20098.63} C_VEL
LIN {X 0,Y 343.048,Z 601.396,A -85,B 0,C 180,E1 -20101.355,E2 -20101.355} C_VEL
LIN {X 0,Y 339.137,Z 597.688,A -85,B 0,C 180,E1 -20103.274,E2 -20103.274} C_VEL
LIN {X 0,Y 333.984,Z 593.366,A -85,B 0,C 180,E1 -20105.663,E2 -20105.663} C_VEL
LIN {X 0,Y 330.388,Z 590.017,A -85,B 0,C 180,E1 -20107.274,E2 -20107.274} C_VEL
LIN {X 0,Y 325.201,Z 585.313,A -85,B 0,C 180,E1 -20109.517,E2 -20109.517} C_VEL
LIN {X 0,Y 322.737,Z 583.005,A -85,B 0,C 180,E1 -20110.551,E2 -20110.551} C_VEL
LIN {X 0,Y 317.699,Z 578.302,A -85,B 0,C 180,E1 -20112.627,E2 -20112.627} C_VEL
LIN {X 0,Y 311.478,Z 572.595,A -85,B 0,C 180,E1 -20115.025,E2 -20115.025} C_VEL
LIN {X 0,Y 305.89,Z 567.629,A -85,B 0,C 180,E1 -20116.971,E2 -20116.971} C_VEL
LIN {X 0,Y 300.603,Z 562.852,A -85,B 0,C 180,E1 -20118.7,E2 -20118.7} C_VEL
LIN {X 0,Y 294.792,Z 557.631,A -85,B 0,C 180,E1 -20120.485,E2 -20120.485} C_VEL
LIN {X 0,Y 287.856,Z 551.542,A -85,B 0,C 180,E1 -20122.494,E2 -20122.494} C_VEL
LIN {X 0,Y 279.901,Z 543.173,A -85,B 0,C 180,E1 -20125.055,E2 -20125.055} C_VEL
LIN {X 0,Y 274.63,Z 536.679,A -85,B 0,C 180,E1 -20126.98,E2 -20126.98} C_VEL
LIN {X 0,Y 266.573,Z 525.491,A -85,B 0,C 180,E1 -20130.368,E2 -20130.368} C_VEL
LIN {X 0,Y 263.466,Z 521.311,A -85,B 0,C 180,E1 -20131.826,E2 -20131.826} C_VEL
LIN {X 0,Y 260.278,Z 517.076,A -85,B 0,C 180,E1 -20133.435,E2 -20133.435} C_VEL
LIN {X 0,Y 256.78,Z 512.502,A -85,B 0,C 180,E1 -20135.358,E2 -20135.358} C_VEL
LIN {X 0,Y 253.753,Z 508.637,A -85,B 0,C 180,E1 -20137.186,E2 -20137.186} C_VEL
LIN {X 0,Y 250.248,Z 504.872,A -85,B 0,C 180,E1 -20139.501,E2 -20139.501} C_VEL
LIN {X 0,Y 249.064,Z 502.854,A -85,B 0,C 180,E1 -20140.423,E2 -20140.423} C_VEL
LIN {X 0,Y 246.2,Z 500.276,A -85,B 0,C 180,E1 -20142.666,E2 -20142.666} C_VEL
LIN {X 0,Y 244.482,Z 497.309,A -85,B 0,C 180,E1 -20144.342,E2 -20144.342} C_VEL
LIN {X 0,Y 241.547,Z 495.125,A -85,B 0,C 180,E1 -20147.396,E2 -20147.396} C_VEL
LIN {X 0,Y 240.067,Z 492.381,A -85,B 0,C 180,E1 -20149.564,E2 -20149.564} C_VEL
LIN {X 0,Y 239.317,Z 491.403,A -85,B 0,C 180,E1 -20150.796,E2 -20150.796} C_VEL
LIN {X 0,Y 236.686,Z 489.508,A -85,B 0,C 180,E1 -20158.299,E2 -20158.299} C_VEL
LIN {X 0,Y 236.727,Z 489.585,A -85,B 0,C 180,E1 -20161.702,E2 -20161.702} C_VEL
LIN {X 0,Y 239.698,Z 491.732,A -85,B 0,C 180,E1 -20169.404,E2 -20169.404} C_VEL
LIN {X 0,Y 241.793,Z 495.386,A -85,B 0,C 180,E1 -20172.485,E2 -20172.485} C_VEL
LIN {X 0,Y 244.787,Z 497.644,A -85,B 0,C 180,E1 -20175.533,E2 -20175.533} C_VEL
LIN {X 0,Y 246.651,Z 500.774,A -85,B 0,C 180,E1 -20177.302,E2 -20177.302} C_VEL
LIN {X 0,Y 249.37,Z 503.227,A -85,B 0,C 180,E1 -20179.392,E2 -20179.392} C_VEL
LIN {X 0,Y 251.501,Z 506.457,A -85,B 0,C 180,E1 -20180.965,E2 -20180.965} C_VEL
LIN {X 0,Y 253.732,Z 508.632,A -85,B 0,C 180,E1 -20182.387,E2 -20182.387} C_VEL
LIN {X 0,Y 256.635,Z 512.375,A -85,B 0,C 180,E1 -20184.146,E2 -20184.146} C_VEL
LIN {X 0,Y 258.092,Z 514.226,A -85,B 0,C 180,E1 -20184.97,E2 -20184.97} C_VEL
LIN {X 0,Y 261.462,Z 518.6,A -85,B 0,C 180,E1 -20186.759,E2 -20186.759} C_VEL
LIN {X 0,Y 265.309,Z 523.874,A -85,B 0,C 180,E1 -20188.64,E2 -20188.64} C_VEL
LIN {X 0,Y 267.916,Z 527.768,A -85,B 0,C 180,E1 -20189.841,E2 -20189.841} C_VEL
LIN {X 0,Y 273.218,Z 536.855,A -85,B 0,C 180,E1 -20192.151,E2 -20192.151} C_VEL
LIN {X 0,Y 279.432,Z 548.287,A -85,B 0,C 180,E1 -20194.616,E2 -20194.616} C_VEL
LIN {X 0,Y 286.6,Z 563.174,A -85,B 0,C 180,E1 -20197.231,E2 -20197.231} C_VEL
LIN {X 0,Y 290.597,Z 572.364,A -85,B 0,C 180,E1 -20198.605,E2 -20198.605} C_VEL
LIN {X 0,Y 286.372,Z 639.328,A -85,B 0,C 180,E1 -20200.153,E2 -20200.153} C_VEL
LIN {X 0,Y 285.581,Z 645.178,A -85,B 0,C 180,E1 -20200.189,E2 -20200.189} C_VEL
LIN {X 0,Y 280.669,Z 664.273,A -85,B 0,C 180,E1 -20199.747,E2 -20199.747} C_VEL
LIN {X 0,Y 279.834,Z 670.127,A -85,B 0,C 180,E1 -20199.772,E2 -20199.772} C_VEL
LIN {X 0,Y 278.072,Z 692.552,A -85,B 0,C 180,E1 -20200.346,E2 -20200.346} C_VEL
LIN {X 0,Y 275.592,Z 709.75,A -85,B 0,C 180,E1 -20201.004,E2 -20201.004} C_VEL
LIN {X 0,Y 272.998,Z 723.384,A -85,B 0,C 180,E1 -20201.707,E2 -20201.707} C_VEL
LIN {X 0,Y 270.057,Z 736.252,A -85,B 0,C 180,E1 -20202.55,E2 -20202.55} C_VEL
LIN {X 0,Y 266.736,Z 748.818,A -85,B 0,C 180,E1 -20203.568,E2 -20203.568} C_VEL
LIN {X 0,Y 263.242,Z 760.454,A -85,B 0,C 180,E1 -20204.699,E2 -20204.699} C_VEL
LIN {X 0,Y 258.94,Z 773.28,A -85,B 0,C 180,E1 -20206.204,E2 -20206.204} C_VEL
LIN {X 0,Y 254.725,Z 784.407,A -85,B 0,C 180,E1 -20207.739,E2 -20207.739} C_VEL
LIN {X 0,Y 250.655,Z 794.67,A -85,B 0,C 180,E1 -20209.43,E2 -20209.43} C_VEL
LIN {X 0,Y 246.612,Z 803.923,A -85,B 0,C 180,E1 -20211.175,E2 -20211.175} C_VEL
LIN {X 0,Y 242.011,Z 814.129,A -85,B 0,C 180,E1 -20213.466,E2 -20213.466} C_VEL
LIN {X 0,Y 237.811,Z 823.086,A -85,B 0,C 180,E1 -20215.841,E2 -20215.841} C_VEL
LIN {X 0,Y 234.111,Z 830.98,A -85,B 0,C 180,E1 -20218.309,E2 -20218.309} C_VEL
LIN {X 0,Y 230.651,Z 837.942,A -85,B 0,C 180,E1 -20220.823,E2 -20220.823} C_VEL
LIN {X 0,Y 227.529,Z 844.477,A -85,B 0,C 180,E1 -20223.606,E2 -20223.606} C_VEL
LIN {X 0,Y 224.525,Z 851.037,A -85,B 0,C 180,E1 -20226.967,E2 -20226.967} C_VEL
LIN {X 0,Y 222.06,Z 856.801,A -85,B 0,C 180,E1 -20230.591,E2 -20230.591} C_VEL
LIN {X 0,Y 220.718,Z 860.423,A -85,B 0,C 180,E1 -20233.347,E2 -20233.347} C_VEL
LIN {X 0,Y 219.344,Z 864.28,A -85,B 0,C 180,E1 -20237.039,E2 -20237.039} C_VEL
LIN {X 0,Y 218.692,Z 867.143,A -85,B 0,C 180,E1 -20240.754,E2 -20240.754} C_VEL
LIN {X 0,Y 218.539,Z 868.285,A -85,B 0,C 180,E1 -20242.609,E2 -20242.609} C_VEL
LIN {X 0,Y 218.498,Z 869.72,A -85,B 0,C 180,E1 -20246.312,E2 -20246.312} C_VEL
LIN {X 0,Y 218.605,Z 870.2,A -85,B 0,C 180,E1 -20250,E2 -20250} C_VEL
LIN {X 0,Y 218.48,Z 869.5,A -85,B 0,C 180,E1 -20254.292,E2 -20254.292} C_VEL
LIN {X 0,Y 218.539,Z 868.285,A -85,B 0,C 180,E1 -20257.391,E2 -20257.391} C_VEL
LIN {X 0,Y 218.939,Z 865.887,A -85,B 0,C 180,E1 -20261.104,E2 -20261.104} C_VEL
LIN {X 0,Y 220.308,Z 861.464,A -85,B 0,C 180,E1 -20265.733,E2 -20265.733} C_VEL
LIN {X 0,Y 221.548,Z 858.09,A -85,B 0,C 180,E1 -20268.495,E2 -20268.495} C_VEL
LIN {X 0,Y 223.838,Z 852.583,A -85,B 0,C 180,E1 -20272.133,E2 -20272.133} C_VEL
LIN {X 0,Y 226.055,Z 847.72,A -85,B 0,C 180,E1 -20274.816,E2 -20274.816} C_VEL
LIN {X 0,Y 229.613,Z 840.048,A -85,B 0,C 180,E1 -20278.321,E2 -20278.321} C_VEL
LIN {X 0,Y 232.892,Z 833.396,A -85,B 0,C 180,E1 -20280.864,E2 -20280.864} C_VEL
LIN {X 0,Y 236.515,Z 825.956,A -85,B 0,C 180,E1 -20283.306,E2 -20283.306} C_VEL
LIN {X 0,Y 240.556,Z 817.26,A -85,B 0,C 180,E1 -20285.754,E2 -20285.754} C_VEL
LIN {X 0,Y 245.029,Z 807.473,A -85,B 0,C 180,E1 -20288.072,E2 -20288.072} C_VEL
LIN {X 0,Y 249.53,Z 797.257,A -85,B 0,C 180,E1 -20290.11,E2 -20290.11} C_VEL
LIN {X 0,Y 253.848,Z 786.695,A -85,B 0,C 180,E1 -20291.906,E2 -20291.906} C_VEL
LIN {X 0,Y 257.957,Z 775.888,A -85,B 0,C 180,E1 -20293.465,E2 -20293.465} C_VEL
LIN {X 0,Y 261.755,Z 764.952,A -85,B 0,C 180,E1 -20294.812,E2 -20294.812} C_VEL
LIN {X 0,Y 265.251,Z 754.042,A -85,B 0,C 180,E1 -20295.945,E2 -20295.945} C_VEL
LIN {X 0,Y 268.807,Z 741.315,A -85,B 0,C 180,E1 -20297.058,E2 -20297.058} C_VEL
LIN {X 0,Y 271.971,Z 728.235,A -85,B 0,C 180,E1 -20297.99,E2 -20297.99} C_VEL
LIN {X 0,Y 274.653,Z 715.113,A -85,B 0,C 180,E1 -20298.733,E2 -20298.733} C_VEL
LIN {X 0,Y 276.864,Z 701.747,A -85,B 0,C 180,E1 -20299.318,E2 -20299.318} C_VEL
LIN {X 0,Y 278.455,Z 688.294,A -85,B 0,C 180,E1 -20299.771,E2 -20299.771} C_VEL
LIN {X 0,Y 281.065,Z 651.009,A -85,B 0,C 180,E1 -20300.676,E2 -20300.676} C_VEL
LIN {X 0,Y 285.99,Z 575.575,A -85,B 0,C 180,E1 -20302.428,E2 -20302.428} C_VEL
LIN {X 0,Y 285.478,Z 573.766,A -85,B 0,C 180,E1 -20302.634,E2 -20302.634} C_VEL
LIN {X 0,Y 278.987,Z 559.236,A -85,B 0,C 180,E1 -20305.033,E2 -20305.033} C_VEL
LIN {X 0,Y 273.46,Z 548.256,A -85,B 0,C 180,E1 -20307.227,E2 -20307.227} C_VEL
LIN {X 0,Y 268.049,Z 538.32,A -85,B 0,C 180,E1 -20309.562,E2 -20309.562} C_VEL
LIN {X 0,Y 263.74,Z 531.089,A -85,B 0,C 180,E1 -20311.581,E2 -20311.581} C_VEL
LIN {X 0,Y 260.842,Z 527,A -85,B 0,C 180,E1 -20313.01,E2 -20313.01} C_VEL
LIN {X 0,Y 258.003,Z 523.141,A -85,B 0,C 180,E1 -20314.506,E2 -20314.506} C_VEL
LIN {X 0,Y 254.822,Z 518.929,A -85,B 0,C 180,E1 -20316.319,E2 -20316.319} C_VEL
LIN {X 0,Y 251.911,Z 515.112,A -85,B 0,C 180,E1 -20318.144,E2 -20318.144} C_VEL
LIN {X 0,Y 248.391,Z 511.052,A -85,B 0,C 180,E1 -20320.582,E2 -20320.582} C_VEL
LIN {X 0,Y 247.421,Z 509.429,A -85,B 0,C 180,E1 -20321.364,E2 -20321.364} C_VEL
LIN {X 0,Y 244.649,Z 506.725,A -85,B 0,C 180,E1 -20323.64,E2 -20323.64} C_VEL
LIN {X 0,Y 243.171,Z 504.15,A -85,B 0,C 180,E1 -20325.137,E2 -20325.137} C_VEL
LIN {X 0,Y 240.43,Z 502.021,A -85,B 0,C 180,E1 -20328.086,E2 -20328.086} C_VEL
LIN {X 0,Y 238.954,Z 499.293,A -85,B 0,C 180,E1 -20330.319,E2 -20330.319} C_VEL
LIN {X 0,Y 238.473,Z 498.495,A -85,B 0,C 180,E1 -20331.155,E2 -20331.155} C_VEL
LIN {X 0,Y 235.758,Z 496.422,A -85,B 0,C 180,E1 -20340,E2 -20340} C_VEL
LIN {X 0,Y 236.245,Z 497.262,A -85,B 0,C 180,E1 -20344.265,E2 -20344.265} C_VEL
LIN {X 0,Y 238.7,Z 498.74,A -85,B 0,C 180,E1 -20349.642,E2 -20349.642} C_VEL
LIN {X 0,Y 240.359,Z 501.934,A -85,B 0,C 180,E1 -20352.238,E2 -20352.238} C_VEL
LIN {X 0,Y 243.37,Z 504.413,A -85,B 0,C 180,E1 -20355.481,E2 -20355.481} C_VEL
LIN {X 0,Y 245.336,Z 507.645,A -85,B 0,C 180,E1 -20357.397,E2 -20357.397} C_VEL
LIN {X 0,Y 247.733,Z 509.969,A -85,B 0,C 180,E1 -20359.309,E2 -20359.309} C_VEL
LIN {X 0,Y 250.272,Z 513.519,A -85,B 0,C 180,E1 -20361.203,E2 -20361.203} C_VEL
LIN {X 0,Y 252.071,Z 515.357,A -85,B 0,C 180,E1 -20362.38,E2 -20362.38} C_VEL
LIN {X 0,Y 255.915,Z 520.342,A -85,B 0,C 180,E1 -20364.737,E2 -20364.737} C_VEL
LIN {X 0,Y 259.703,Z 525.437,A -85,B 0,C 180,E1 -20366.818,E2 -20366.818} C_VEL
LIN {X 0,Y 265.225,Z 532.943,A -85,B 0,C 180,E1 -20369.518,E2 -20369.518} C_VEL
LIN {X 0,Y 276.083,Z 547.912,A -85,B 0,C 180,E1 -20374.003,E2 -20374.003} C_VEL
LIN {X 0,Y 282.597,Z 555.067,A -85,B 0,C 180,E1 -20376.232,E2 -20376.232} C_VEL
LIN {X 0,Y 290.271,Z 562.34,A -85,B 0,C 180,E1 -20378.551,E2 -20378.551} C_VEL
LIN {X 0,Y 298.34,Z 569.312,A -85,B 0,C 180,E1 -20380.932,E2 -20380.932} C_VEL
LIN {X 0,Y 305.195,Z 575.36,A -85,B 0,C 180,E1 -20383.163,E2 -20383.163} C_VEL
LIN {X 0,Y 309.045,Z 578.77,A -85,B 0,C 180,E1 -20384.498,E2 -20384.498} C_VEL
LIN {X 0,Y 314.188,Z 583.299,A -85,B 0,C 180,E1 -20386.384,E2 -20386.384} C_VEL
LIN {X 0,Y 320.224,Z 589.036,A -85,B 0,C 180,E1 -20388.822,E2 -20388.822} C_VEL
LIN {X 0,Y 324.012,Z 592.47,A -85,B 0,C 180,E1 -20390.401,E2 -20390.401} C_VEL
LIN {X 0,Y 328.972,Z 596.899,A -85,B 0,C 180,E1 -20392.533,E2 -20392.533} C_VEL
LIN {X 0,Y 335.179,Z 602.571,A -85,B 0,C 180,E1 -20395.329,E2 -20395.329} C_VEL
LIN {X 0,Y 339.31,Z 605.942,A -85,B 0,C 180,E1 -20397.266,E2 -20397.266} C_VEL
LIN {X 0,Y 343.554,Z 609.787,A -85,B 0,C 180,E1 -20399.372,E2 -20399.372} C_VEL
LIN {X 0,Y 347.134,Z 612.608,A -85,B 0,C 180,E1 -20401.216,E2 -20401.216} C_VEL
LIN {X 0,Y 351.458,Z 616.737,A -85,B 0,C 180,E1 -20403.638,E2 -20403.638} C_VEL
LIN {X 0,Y 356.049,Z 620.035,A -85,B 0,C 180,E1 -20406.357,E2 -20406.357} C_VEL
LIN {X 0,Y 359.334,Z 623.214,A -85,B 0,C 180,E1 -20408.535,E2 -20408.535} C_VEL
LIN {X 0,Y 362.895,Z 625.785,A -85,B 0,C 180,E1 -20411.104,E2 -20411.104} C_VEL
LIN {X 0,Y 365.26,Z 627.25,A -85,B 0,C 180,E1 -20412.956,E2 -20412.956} C_VEL
LIN {X 0,Y 367.876,Z 630.063,A -85,B 0,C 180,E1 -20415.425,E2 -20415.425} C_VEL
LIN {X 0,Y 370.237,Z 632.007,A -85,B 0,C 180,E1 -20417.948,E2 -20417.948} C_VEL
LIN {X 0,Y 372.25,Z 633.095,A -85,B 0,C 180,E1 -20420.562,E2 -20420.562} C_VEL
LIN {X 0,Y 373.655,Z 633.793,A -85,B 0,C 180,E1 -20422.847,E2 -20422.847} C_VEL
LIN {X 0,Y 374.664,Z 634.413,A -85,B 0,C 180,E1 -20425.186,E2 -20425.186} C_VEL
LIN {X 0,Y 375.366,Z 634.657,A -85,B 0,C 180,E1 -20427.854,E2 -20427.854} C_VEL
LIN {X 0,Y 375.553,Z 634.763,A -85,B 0,C 180,E1 -20430,E2 -20430} C_VEL
LIN {X 0,Y 375.366,Z 634.656,A -85,B 0,C 180,E1 -20432.146,E2 -20432.146} C_VEL
LIN {X 0,Y 374.665,Z 634.407,A -85,B 0,C 180,E1 -20434.815,E2 -20434.815} C_VEL
LIN {X 0,Y 373.418,Z 633.644,A -85,B 0,C 180,E1 -20437.57,E2 -20437.57} C_VEL
LIN {X 0,Y 371.573,Z 632.783,A -85,B 0,C 180,E1 -20440.414,E2 -20440.414} C_VEL
LIN {X 0,Y 369.365,Z 631.333,A -85,B 0,C 180,E1 -20443.017,E2 -20443.017} C_VEL
LIN {X 0,Y 366.878,Z 629.056,A -85,B 0,C 180,E1 -20445.556,E2 -20445.556} C_VEL
LIN {X 0,Y 364.481,Z 626.66,A -85,B 0,C 180,E1 -20447.676,E2 -20447.676} C_VEL
LIN {X 0,Y 361.28,Z 624.674,A -85,B 0,C 180,E1 -20450.097,E2 -20450.097} C_VEL
LIN {X 0,Y 357.7,Z 621.768,A -85,B 0,C 180,E1 -20452.567,E2 -20452.567} C_VEL
LIN {X 0,Y 355.071,Z 619.188,A -85,B 0,C 180,E1 -20454.27,E2 -20454.27} C_VEL
LIN {X 0,Y 351.105,Z 616.436,A -85,B 0,C 180,E1 -20456.567,E2 -20456.567} C_VEL
LIN {X 0,Y 346.886,Z 612.374,A -85,B 0,C 180,E1 -20458.917,E2 -20458.917} C_VEL
LIN {X 0,Y 341.576,Z 608.166,A -85,B 0,C 180,E1 -20461.611,E2 -20461.611} C_VEL
LIN {X 0,Y 337.513,Z 604.359,A -85,B 0,C 180,E1 -20463.602,E2 -20463.602} C_VEL
LIN {X 0,Y 332.302,Z 600.01,A -85,B 0,C 180,E1 -20465.983,E2 -20465.983} C_VEL
LIN {X 0,Y 328.507,Z 596.51,A -85,B 0,C 180,E1 -20467.669,E2 -20467.669} C_VEL
LIN {X 0,Y 323.352,Z 591.853,A -85,B 0,C 180,E1 -20469.876,E2 -20469.876} C_VEL
LIN {X 0,Y 316.443,Z 585.534,A -85,B 0,C 180,E1 -20472.72,E2 -20472.72} C_VEL
LIN {X 0,Y 312.752,Z 582.079,A -85,B 0,C 180,E1 -20474.155,E2 -20474.155} C_VEL
LIN {X 0,Y 307.468,Z 577.166,A -85,B 0,C 180,E1 -20476.084,E2 -20476.084} C_VEL
LIN {X 0,Y 301.336,Z 571.909,A -85,B 0,C 180,E1 -20478.111,E2 -20478.111} C_VEL
LIN {X 0,Y 293.689,Z 565.318,A -85,B 0,C 180,E1 -20480.464,E2 -20480.464} C_VEL
LIN {X 0,Y 284.905,Z 557.38,A -85,B 0,C 180,E1 -20483.039,E2 -20483.039} C_VEL
LIN {X 0,Y 277.292,Z 549.308,A -85,B 0,C 180,E1 -20485.563,E2 -20485.563} C_VEL
LIN {X 0,Y 271.732,Z 542.276,A -85,B 0,C 180,E1 -20487.667,E2 -20487.667} C_VEL
LIN {X 0,Y 264.101,Z 531.494,A -85,B 0,C 180,E1 -20491,E2 -20491} C_VEL
LIN {X 0,Y 260.454,Z 526.499,A -85,B 0,C 180,E1 -20492.791,E2 -20492.791} C_VEL
LIN {X 0,Y 258.042,Z 523.197,A -85,B 0,C 180,E1 -20494.068,E2 -20494.068} C_VEL
LIN {X 0,Y 254.849,Z 518.919,A -85,B 0,C 180,E1 -20495.891,E2 -20495.891} C_VEL
LIN {X 0,Y 251.421,Z 514.565,A -85,B 0,C 180,E1 -20498.046,E2 -20498.046} C_VEL
LIN {X 0,Y 248.556,Z 511.387,A -85,B 0,C 180,E1 -20500.031,E2 -20500.031} C_VEL
LIN {X 0,Y 247.428,Z 509.527,A -85,B 0,C 180,E1 -20500.935,E2 -20500.935} C_VEL
LIN {X 0,Y 244.561,Z 506.665,A -85,B 0,C 180,E1 -20503.3,E2 -20503.3} C_VEL
LIN {X 0,Y 243.133,Z 504.154,A -85,B 0,C 180,E1 -20504.754,E2 -20504.754} C_VEL
LIN {X 0,Y 240.36,Z 501.927,A -85,B 0,C 180,E1 -20507.762,E2 -20507.762} C_VEL
LIN {X 0,Y 238.891,Z 499.171,A -85,B 0,C 180,E1 -20510.011,E2 -20510.011} C_VEL
LIN {X 0,Y 238.234,Z 498.341,A -85,B 0,C 180,E1 -20511.136,E2 -20511.136} C_VEL
LIN {X 0,Y 235.821,Z 496.553,A -85,B 0,C 180,E1 -20518.293,E2 -20518.293} C_VEL
LIN {X 0,Y 235.862,Z 496.64,A -85,B 0,C 180,E1 -20521.708,E2 -20521.708} C_VEL
LIN {X 0,Y 238.579,Z 498.591,A -85,B 0,C 180,E1 -20529.021,E2 -20529.021} C_VEL
LIN {X 0,Y 240.676,Z 502.31,A -85,B 0,C 180,E1 -20532.223,E2 -20532.223} C_VEL
LIN {X 0,Y 243.466,Z 504.589,A -85,B 0,C 180,E1 -20535.166,E2 -20535.166} C_VEL
LIN {X 0,Y 245.44,Z 507.735,A -85,B 0,C 180,E1 -20537.068,E2 -20537.068} C_VEL
LIN {X 0,Y 247.791,Z 509.936,A -85,B 0,C 180,E1 -20538.929,E2 -20538.929} C_VEL
LIN {X 0,Y 250.151,Z 513.357,A -85,B 0,C 180,E1 -20540.702,E2 -20540.702} C_VEL
LIN {X 0,Y 252.013,Z 515.3,A -85,B 0,C 180,E1 -20541.928,E2 -20541.928} C_VEL
LIN {X 0,Y 255.143,Z 519.252,A -85,B 0,C 180,E1 -20543.865,E2 -20543.865} C_VEL
LIN {X 0,Y 259.589,Z 525.305,A -85,B 0,C 180,E1 -20546.344,E2 -20546.344} C_VEL
LIN {X 0,Y 263.038,Z 530.099,A -85,B 0,C 180,E1 -20548.082,E2 -20548.082} C_VEL
LIN {X 0,Y 265.214,Z 533.449,A -85,B 0,C 180,E1 -20549.125,E2 -20549.125} C_VEL
LIN {X 0,Y 270.026,Z 541.84,A -85,B 0,C 180,E1 -20551.314,E2 -20551.314} C_VEL
LIN {X 0,Y 276.198,Z 553.496,A -85,B 0,C 180,E1 -20553.877,E2 -20553.877} C_VEL
LIN {X 0,Y 282.361,Z 566.633,A -85,B 0,C 180,E1 -20556.238,E2 -20556.238} C_VEL
LIN {X 0,Y 285.928,Z 574.833,A -85,B 0,C 180,E1 -20557.526,E2 -20557.526} C_VEL
LIN {X 0,Y 282.135,Z 635.276,A -85,B 0,C 180,E1 -20558.97,E2 -20558.97} C_VEL
LIN {X 0,Y 279.834,Z 670.127,A -85,B 0,C 180,E1 -20559.772,E2 -20559.772} C_VEL
LIN {X 0,Y 278.985,Z 675.977,A -85,B 0,C 180,E1 -20559.791,E2 -20559.791} C_VEL
LIN {X 0,Y 273.554,Z 694.959,A -85,B 0,C 180,E1 -20559.386,E2 -20559.386} C_VEL
LIN {X 0,Y 272.376,Z 700.728,A -85,B 0,C 180,E1 -20559.512,E2 -20559.512} C_VEL
LIN {X 0,Y 270.141,Z 714.136,A -85,B 0,C 180,E1 -20560.091,E2 -20560.091} C_VEL
LIN {X 0,Y 267.4,Z 727.246,A -85,B 0,C 180,E1 -20560.821,E2 -20560.821} C_VEL
LIN {X 0,Y 264.431,Z 739.441,A -85,B 0,C 180,E1 -20561.681,E2 -20561.681} C_VEL
LIN {X 0,Y 260.843,Z 752.09,A -85,B 0,C 180,E1 -20562.761,E2 -20562.761} C_VEL
LIN {X 0,Y 256.746,Z 764.741,A -85,B 0,C 180,E1 -20564.067,E2 -20564.067} C_VEL
LIN {X 0,Y 251.375,Z 779.583,A -85,B 0,C 180,E1 -20565.937,E2 -20565.937} C_VEL
LIN {X 0,Y 245.58,Z 793.686,A -85,B 0,C 180,E1 -20568.198,E2 -20568.198} C_VEL
LIN {X 0,Y 241.074,Z 803.712,A -85,B 0,C 180,E1 -20570.108,E2 -20570.108} C_VEL
LIN {X 0,Y 236.271,Z 813.916,A -85,B 0,C 180,E1 -20572.427,E2 -20572.427} C_VEL
LIN {X 0,Y 231.882,Z 822.873,A -85,B 0,C 180,E1 -20574.841,E2 -20574.841} C_VEL
LIN {X 0,Y 228.022,Z 830.767,A -85,B 0,C 180,E1 -20577.36,E2 -20577.36} C_VEL
LIN {X 0,Y 224.403,Z 837.729,A -85,B 0,C 180,E1 -20579.928,E2 -20579.928} C_VEL
LIN {X 0,Y 220.85,Z 844.724,A -85,B 0,C 180,E1 -20583.003,E2 -20583.003} C_VEL
LIN {X 0,Y 217.897,Z 850.823,A -85,B 0,C 180,E1 -20586.224,E2 -20586.224} C_VEL
LIN {X 0,Y 215.274,Z 856.588,A -85,B 0,C 180,E1 -20589.953,E2 -20589.953} C_VEL
LIN {X 0,Y 213.82,Z 860.209,A -85,B 0,C 180,E1 -20592.794,E2 -20592.794} C_VEL
LIN {X 0,Y 212.371,Z 864.069,A -85,B 0,C 180,E1 -20596.606,E2 -20596.606} C_VEL
LIN {X 0,Y 211.619,Z 866.931,A -85,B 0,C 180,E1 -20600.442,E2 -20600.442} C_VEL
LIN {X 0,Y 211.448,Z 868.073,A -85,B 0,C 180,E1 -20602.36,E2 -20602.36} C_VEL
LIN {X 0,Y 211.396,Z 869.51,A -85,B 0,C 180,E1 -20606.188,E2 -20606.188} C_VEL
LIN {X 0,Y 211.523,Z 869.991,A -85,B 0,C 180,E1 -20610,E2 -20610} C_VEL
LIN {X 0,Y 211.393,Z 869.393,A -85,B 0,C 180,E1 -20614.145,E2 -20614.145} C_VEL
LIN {X 0,Y 211.448,Z 868.073,A -85,B 0,C 180,E1 -20617.64,E2 -20617.64} C_VEL
LIN {X 0,Y 211.894,Z 865.675,A -85,B 0,C 180,E1 -20621.479,E2 -20621.479} C_VEL
LIN {X 0,Y 213.404,Z 861.251,A -85,B 0,C 180,E1 -20626.256,E2 -20626.256} C_VEL
LIN {X 0,Y 214.734,Z 857.877,A -85,B 0,C 180,E1 -20629.104,E2 -20629.104} C_VEL
LIN {X 0,Y 217.158,Z 852.369,A -85,B 0,C 180,E1 -20632.852,E2 -20632.852} C_VEL
LIN {X 0,Y 219.496,Z 847.506,A -85,B 0,C 180,E1 -20635.61,E2 -20635.61} C_VEL
LIN {X 0,Y 223.272,Z 839.834,A -85,B 0,C 180,E1 -20639.202,E2 -20639.202} C_VEL
LIN {X 0,Y 226.735,Z 833.183,A -85,B 0,C 180,E1 -20641.798,E2 -20641.798} C_VEL
LIN {X 0,Y 230.342,Z 826.086,A -85,B 0,C 180,E1 -20644.19,E2 -20644.19} C_VEL
LIN {X 0,Y 234.75,Z 817.047,A -85,B 0,C 180,E1 -20646.781,E2 -20646.781} C_VEL
LIN {X 0,Y 239.398,Z 807.26,A -85,B 0,C 180,E1 -20649.136,E2 -20649.136} C_VEL
LIN {X 0,Y 244.098,Z 797.045,A -85,B 0,C 180,E1 -20651.193,E2 -20651.193} C_VEL
LIN {X 0,Y 248.547,Z 786.482,A -85,B 0,C 180,E1 -20653.012,E2 -20653.012} C_VEL
LIN {X 0,Y 252.795,Z 775.675,A -85,B 0,C 180,E1 -20654.585,E2 -20654.585} C_VEL
LIN {X 0,Y 256.743,Z 764.741,A -85,B 0,C 180,E1 -20655.934,E2 -20655.934} C_VEL
LIN {X 0,Y 260.338,Z 753.831,A -85,B 0,C 180,E1 -20657.074,E2 -20657.074} C_VEL
LIN {X 0,Y 264.257,Z 740.089,A -85,B 0,C 180,E1 -20658.27,E2 -20658.27} C_VEL
LIN {X 0,Y 267.14,Z 728.605,A -85,B 0,C 180,E1 -20659.086,E2 -20659.086} C_VEL
LIN {X 0,Y 270.026,Z 714.904,A -85,B 0,C 180,E1 -20659.865,E2 -20659.865} C_VEL
LIN {X 0,Y 272.288,Z 701.537,A -85,B 0,C 180,E1 -20660.451,E2 -20660.451} C_VEL
LIN {X 0,Y 273.926,Z 688.084,A -85,B 0,C 180,E1 -20660.904,E2 -20660.904} C_VEL
LIN {X 0,Y 276.615,Z 650.799,A -85,B 0,C 180,E1 -20661.815,E2 -20661.815} C_VEL
LIN {X 0,Y 281.529,Z 577.705,A -85,B 0,C 180,E1 -20663.526,E2 -20663.526} C_VEL
LIN {X 0,Y 274.696,Z 562.2,A -85,B 0,C 180,E1 -20666.188,E2 -20666.188} C_VEL
LIN {X 0,Y 268.67,Z 550.219,A -85,B 0,C 180,E1 -20668.737,E2 -20668.737} C_VEL
LIN {X 0,Y 263.674,Z 541.048,A -85,B 0,C 180,E1 -20671.057,E2 -20671.057} C_VEL
LIN {X 0,Y 260.927,Z 536.529,A -85,B 0,C 180,E1 -20672.418,E2 -20672.418} C_VEL
LIN {X 0,Y 256.339,Z 529.93,A -85,B 0,C 180,E1 -20674.851,E2 -20674.851} C_VEL
LIN {X 0,Y 252.872,Z 525.312,A -85,B 0,C 180,E1 -20676.885,E2 -20676.885} C_VEL
LIN {X 0,Y 249.612,Z 521.052,A -85,B 0,C 180,E1 -20679.016,E2 -20679.016} C_VEL
LIN {X 0,Y 246.607,Z 517.348,A -85,B 0,C 180,E1 -20681.219,E2 -20681.219} C_VEL
LIN {X 0,Y 245.808,Z 516.061,A -85,B 0,C 180,E1 -20681.884,E2 -20681.884} C_VEL
LIN {X 0,Y 243.178,Z 513.299,A -85,B 0,C 180,E1 -20684.145,E2 -20684.145} C_VEL
LIN {X 0,Y 241.901,Z 511.046,A -85,B 0,C 180,E1 -20685.488,E2 -20685.488} C_VEL
LIN {X 0,Y 239.017,Z 508.549,A -85,B 0,C 180,E1 -20688.767,E2 -20688.767} C_VEL
LIN {X 0,Y 237.521,Z 505.512,A -85,B 0,C 180,E1 -20691.275,E2 -20691.275} C_VEL
LIN {X 0,Y 234.999,Z 503.67,A -85,B 0,C 180,E1 -20698.286,E2 -20698.286} C_VEL
LIN {X 0,Y 234.952,Z 503.638,A -85,B 0,C 180,E1 -20701.714,E2 -20701.714} C_VEL
LIN {X 0,Y 237.661,Z 505.696,A -85,B 0,C 180,E1 -20709.387,E2 -20709.387} C_VEL
LIN {X 0,Y 239.255,Z 508.862,A -85,B 0,C 180,E1 -20711.973,E2 -20711.973} C_VEL
LIN {X 0,Y 242.027,Z 511.286,A -85,B 0,C 180,E1 -20715.069,E2 -20715.069} C_VEL
LIN {X 0,Y 244.245,Z 514.752,A -85,B 0,C 180,E1 -20717.261,E2 -20717.261} C_VEL
LIN {X 0,Y 246.233,Z 516.769,A -85,B 0,C 180,E1 -20718.891,E2 -20718.891} C_VEL
LIN {X 0,Y 248.884,Z 520.387,A -85,B 0,C 180,E1 -20720.91,E2 -20720.91} C_VEL
LIN {X 0,Y 250.406,Z 522.052,A -85,B 0,C 180,E1 -20721.939,E2 -20721.939} C_VEL
LIN {X 0,Y 253.963,Z 526.724,A -85,B 0,C 180,E1 -20724.192,E2 -20724.192} C_VEL
LIN {X 0,Y 257.775,Z 532.018,A -85,B 0,C 180,E1 -20726.36,E2 -20726.36} C_VEL
LIN {X 0,Y 262.769,Z 538.971,A -85,B 0,C 180,E1 -20728.887,E2 -20728.887} C_VEL
LIN {X 0,Y 273.408,Z 553.917,A -85,B 0,C 180,E1 -20733.439,E2 -20733.439} C_VEL
LIN {X 0,Y 280.222,Z 561.468,A -85,B 0,C 180,E1 -20735.836,E2 -20735.836} C_VEL
LIN {X 0,Y 287.675,Z 568.625,A -85,B 0,C 180,E1 -20738.143,E2 -20738.143} C_VEL
LIN {X 0,Y 295.449,Z 575.32,A -85,B 0,C 180,E1 -20740.418,E2 -20740.418} C_VEL
LIN {X 0,Y 300.306,Z 579.549,A -85,B 0,C 180,E1 -20741.925,E2 -20741.925} C_VEL
LIN {X 0,Y 307.246,Z 585.5,A -85,B 0,C 180,E1 -20744.233,E2 -20744.233} C_VEL
LIN {X 0,Y 312.473,Z 590.043,A -85,B 0,C 180,E1 -20746.127,E2 -20746.127} C_VEL
LIN {X 0,Y 318.019,Z 595.333,A -85,B 0,C 180,E1 -20748.337,E2 -20748.337} C_VEL
LIN {X 0,Y 321.976,Z 598.86,A -85,B 0,C 180,E1 -20749.969,E2 -20749.969} C_VEL
LIN {X 0,Y 327.158,Z 603.478,A -85,B 0,C 180,E1 -20752.169,E2 -20752.169} C_VEL
LIN {X 0,Y 333.581,Z 609.267,A -85,B 0,C 180,E1 -20755.032,E2 -20755.032} C_VEL
LIN {X 0,Y 337.804,Z 612.727,A -85,B 0,C 180,E1 -20757.006,E2 -20757.006} C_VEL
LIN {X 0,Y 342.192,Z 616.63,A -85,B 0,C 180,E1 -20759.153,E2 -20759.153} C_VEL
LIN {X 0,Y 345.799,Z 619.507,A -85,B 0,C 180,E1 -20761.009,E2 -20761.009} C_VEL
LIN {X 0,Y 350.142,Z 623.574,A -85,B 0,C 180,E1 -20763.411,E2 -20763.411} C_VEL
LIN {X 0,Y 354.808,Z 626.904,A -85,B 0,C 180,E1 -20766.144,E2 -20766.144} C_VEL
LIN {X 0,Y 358.331,Z 630.251,A -85,B 0,C 180,E1 -20768.472,E2 -20768.472} C_VEL
LIN {X 0,Y 361.932,Z 632.821,A -85,B 0,C 180,E1 -20771.052,E2 -20771.052} C_VEL
LIN {X 0,Y 364.305,Z 634.334,A -85,B 0,C 180,E1 -20772.91,E2 -20772.91} C_VEL
LIN {X 0,Y 366.956,Z 637.122,A -85,B 0,C 180,E1 -20775.388,E2 -20775.388} C_VEL
LIN {X 0,Y 369.33,Z 639.055,A -85,B 0,C 180,E1 -20777.918,E2 -20777.918} C_VEL
LIN {X 0,Y 371.362,Z 640.14,A -85,B 0,C 180,E1 -20780.539,E2 -20780.539} C_VEL
LIN {X 0,Y 372.777,Z 640.837,A -85,B 0,C 180,E1 -20782.831,E2 -20782.831} C_VEL
LIN {X 0,Y 373.8,Z 641.444,A -85,B 0,C 180,E1 -20785.184,E2 -20785.184} C_VEL
LIN {X 0,Y 374.501,Z 641.676,A -85,B 0,C 180,E1 -20787.849,E2 -20787.849} C_VEL
LIN {X 0,Y 374.688,Z 641.809,A -85,B 0,C 180,E1 -20790,E2 -20790} C_VEL
LIN {X 0,Y 374.501,Z 641.675,A -85,B 0,C 180,E1 -20792.151,E2 -20792.151} C_VEL
LIN {X 0,Y 373.799,Z 641.447,A -85,B 0,C 180,E1 -20794.816,E2 -20794.816} C_VEL
LIN {X 0,Y 372.536,Z 640.69,A -85,B 0,C 180,E1 -20797.588,E2 -20797.588} C_VEL
LIN {X 0,Y 370.676,Z 639.824,A -85,B 0,C 180,E1 -20800.44,E2 -20800.44} C_VEL
LIN {X 0,Y 368.459,Z 638.384,A -85,B 0,C 180,E1 -20803.049,E2 -20803.049} C_VEL
LIN {X 0,Y 365.94,Z 636.131,A -85,B 0,C 180,E1 -20805.597,E2 -20805.597} C_VEL
LIN {X 0,Y 363.371,Z 633.587,A -85,B 0,C 180,E1 -20807.861,E2 -20807.861} C_VEL
LIN {X 0,Y 360.08,Z 631.561,A -85,B 0,C 180,E1 -20810.303,E2 -20810.303} C_VEL
LIN {X 0,Y 356.434,Z 628.587,A -85,B 0,C 180,E1 -20812.808,E2 -20812.808} C_VEL
LIN {X 0,Y 353.86,Z 626.106,A -85,B 0,C 180,E1 -20814.444,E2 -20814.444} C_VEL
LIN {X 0,Y 349.669,Z 623.17,A -85,B 0,C 180,E1 -20816.868,E2 -20816.868} C_VEL
LIN {X 0,Y 345.347,Z 619.036,A -85,B 0,C 180,E1 -20819.236,E2 -20819.236} C_VEL
LIN {X 0,Y 340.195,Z 615.025,A -85,B 0,C 180,E1 -20821.824,E2 -20821.824} C_VEL
LIN {X 0,Y 335.892,Z 611.06,A -85,B 0,C 180,E1 -20823.904,E2 -20823.904} C_VEL
LIN {X 0,Y 330.567,Z 606.602,A -85,B 0,C 180,E1 -20826.327,E2 -20826.327} C_VEL
LIN {X 0,Y 326.929,Z 603.283,A -85,B 0,C 180,E1 -20827.932,E2 -20827.932} C_VEL
LIN {X 0,Y 321.503,Z 598.413,A -85,B 0,C 180,E1 -20830.23,E2 -20830.23} C_VEL
LIN {X 0,Y 314.784,Z 592.361,A -85,B 0,C 180,E1 -20832.962,E2 -20832.962} C_VEL
LIN {X 0,Y 310.926,Z 588.776,A -85,B 0,C 180,E1 -20834.452,E2 -20834.452} C_VEL
LIN {X 0,Y 304.174,Z 582.766,A -85,B 0,C 180,E1 -20836.814,E2 -20836.814} C_VEL
LIN {X 0,Y 298.872,Z 578.164,A -85,B 0,C 180,E1 -20838.536,E2 -20838.536} C_VEL
LIN {X 0,Y 291.318,Z 571.749,A -85,B 0,C 180,E1 -20840.809,E2 -20840.809} C_VEL
LIN {X 0,Y 282.207,Z 563.517,A -85,B 0,C 180,E1 -20843.52,E2 -20843.52} C_VEL
LIN {X 0,Y 274.49,Z 555.164,A -85,B 0,C 180,E1 -20846.16,E2 -20846.16} C_VEL
LIN {X 0,Y 269.063,Z 548.174,A -85,B 0,C 180,E1 -20848.287,E2 -20848.287} C_VEL
LIN {X 0,Y 261.57,Z 537.346,A -85,B 0,C 180,E1 -20851.689,E2 -20851.689} C_VEL
LIN {X 0,Y 258.206,Z 532.646,A -85,B 0,C 180,E1 -20853.407,E2 -20853.407} C_VEL
LIN {X 0,Y 255.621,Z 529.083,A -85,B 0,C 180,E1 -20854.832,E2 -20854.832} C_VEL
LIN {X 0,Y 252.737,Z 525.115,A -85,B 0,C 180,E1 -20856.554,E2 -20856.554} C_VEL
LIN {X 0,Y 249.566,Z 521.032,A -85,B 0,C 180,E1 -20858.629,E2 -20858.629} C_VEL
LIN {X 0,Y 246.739,Z 517.618,A -85,B 0,C 180,E1 -20860.691,E2 -20860.691} C_VEL
LIN {X 0,Y 245.817,Z 516.151,A -85,B 0,C 180,E1 -20861.454,E2 -20861.454} C_VEL
LIN {X 0,Y 243.051,Z 513.207,A -85,B 0,C 180,E1 -20863.844,E2 -20863.844} C_VEL
LIN {X 0,Y 241.812,Z 510.977,A -85,B 0,C 180,E1 -20865.16,E2 -20865.16} C_VEL
LIN {X 0,Y 239.102,Z 508.662,A -85,B 0,C 180,E1 -20868.234,E2 -20868.234} C_VEL
LIN {X 0,Y 237.489,Z 505.479,A -85,B 0,C 180,E1 -20870.916,E2 -20870.916} C_VEL
LIN {X 0,Y 234.953,Z 503.63,A -85,B 0,C 180,E1 -20878.286,E2 -20878.286} C_VEL
LIN {X 0,Y 234.924,Z 503.537,A -85,B 0,C 180,E1 -20880.857,E2 -20880.857} C_VEL
LIN {X 0,Y 237.64,Z 505.662,A -85,B 0,C 180,E1 -20888.934,E2 -20888.934} C_VEL
LIN {X 0,Y 239.324,Z 508.946,A -85,B 0,C 180,E1 -20891.648,E2 -20891.648} C_VEL
LIN {X 0,Y 242.09,Z 511.343,A -85,B 0,C 180,E1 -20894.716,E2 -20894.716} C_VEL
LIN {X 0,Y 244.235,Z 514.69,A -85,B 0,C 180,E1 -20896.832,E2 -20896.832} C_VEL
LIN {X 0,Y 246.226,Z 516.66,A -85,B 0,C 180,E1 -20898.461,E2 -20898.461} C_VEL
LIN {X 0,Y 248.985,Z 520.467,A -85,B 0,C 180,E1 -20900.562,E2 -20900.562} C_VEL
LIN {X 0,Y 250.382,Z 522.053,A -85,B 0,C 180,E1 -20901.51,E2 -20901.51} C_VEL
LIN {X 0,Y 254.175,Z 527.077,A -85,B 0,C 180,E1 -20903.907,E2 -20903.907} C_VEL
LIN {X 0,Y 257.575,Z 531.739,A -85,B 0,C 180,E1 -20905.836,E2 -20905.836} C_VEL
LIN {X 0,Y 261.904,Z 537.861,A -85,B 0,C 180,E1 -20908.061,E2 -20908.061} C_VEL
LIN {X 0,Y 267.265,Z 547.549,A -85,B 0,C 180,E1 -20910.63,E2 -20910.63} C_VEL
LIN {X 0,Y 273.229,Z 559.112,A -85,B 0,C 180,E1 -20913.209,E2 -20913.209} C_VEL
LIN {X 0,Y 279.893,Z 573.829,A -85,B 0,C 180,E1 -20915.857,E2 -20915.857} C_VEL
LIN {X 0,Y 281.527,Z 577.722,A -85,B 0,C 180,E1 -20916.474,E2 -20916.474} C_VEL
LIN {X 0,Y 274.472,Z 682.508,A -85,B 0,C 180,E1 -20918.945,E2 -20918.945} C_VEL
LIN {X 0,Y 272.834,Z 697.54,A -85,B 0,C 180,E1 -20919.398,E2 -20919.398} C_VEL
LIN {X 0,Y 272.376,Z 700.728,A -85,B 0,C 180,E1 -20919.512,E2 -20919.512} C_VEL
LIN {X 0,Y 271.581,Z 704.563,A -85,B 0,C 180,E1 -20919.589,E2 -20919.589} C_VEL
LIN {X 0,Y 269.041,Z 712.053,A -85,B 0,C 180,E1 -20919.606,E2 -20919.606} C_VEL
LIN {X 0,Y 263.707,Z 724.865,A -85,B 0,C 180,E1 -20919.614,E2 -20919.614} C_VEL
LIN {X 0,Y 262.056,Z 730.422,A -85,B 0,C 180,E1 -20919.862,E2 -20919.862} C_VEL
LIN {X 0,Y 257.516,Z 747.125,A -85,B 0,C 180,E1 -20921.15,E2 -20921.15} C_VEL
LIN {X 0,Y 253.393,Z 760.032,A -85,B 0,C 180,E1 -20922.401,E2 -20922.401} C_VEL
LIN {X 0,Y 248.773,Z 772.855,A -85,B 0,C 180,E1 -20923.915,E2 -20923.915} C_VEL
LIN {X 0,Y 244.328,Z 783.985,A -85,B 0,C 180,E1 -20925.483,E2 -20925.483} C_VEL
LIN {X 0,Y 239.878,Z 794.33,A -85,B 0,C 180,E1 -20927.212,E2 -20927.212} C_VEL
LIN {X 0,Y 235.635,Z 803.501,A -85,B 0,C 180,E1 -20928.993,E2 -20928.993} C_VEL
LIN {X 0,Y 230.602,Z 813.703,A -85,B 0,C 180,E1 -20931.336,E2 -20931.336} C_VEL
LIN {X 0,Y 226.018,Z 822.659,A -85,B 0,C 180,E1 -20933.787,E2 -20933.787} C_VEL
LIN {X 0,Y 221.984,Z 830.554,A -85,B 0,C 180,E1 -20936.356,E2 -20936.356} C_VEL
LIN {X 0,Y 218.177,Z 837.516,A -85,B 0,C 180,E1 -20938.977,E2 -20938.977} C_VEL
LIN {X 0,Y 214.149,Z 845.025,A -85,B 0,C 180,E1 -20942.387,E2 -20942.387} C_VEL
LIN {X 0,Y 211.318,Z 850.61,A -85,B 0,C 180,E1 -20945.436,E2 -20945.436} C_VEL
LIN {X 0,Y 208.507,Z 856.375,A -85,B 0,C 180,E1 -20949.273,E2 -20949.273} C_VEL
LIN {X 0,Y 206.53,Z 861.039,A -85,B 0,C 180,E1 -20953.188,E2 -20953.188} C_VEL
LIN {X 0,Y 204.867,Z 865.463,A -85,B 0,C 180,E1 -20958.122,E2 -20958.122} C_VEL
LIN {X 0,Y 204.379,Z 867.863,A -85,B 0,C 180,E1 -20962.094,E2 -20962.094} C_VEL
LIN {X 0,Y 204.296,Z 869.3,A -85,B 0,C 180,E1 -20966.055,E2 -20966.055} C_VEL
LIN {X 0,Y 204.423,Z 869.781,A -85,B 0,C 180,E1 -20970,E2 -20970} C_VEL
LIN {X 0,Y 204.296,Z 869.3,A -85,B 0,C 180,E1 -20973.945,E2 -20973.945} C_VEL
LIN {X 0,Y 204.378,Z 867.863,A -85,B 0,C 180,E1 -20977.906,E2 -20977.906} C_VEL
LIN {X 0,Y 204.861,Z 865.463,A -85,B 0,C 180,E1 -20981.878,E2 -20981.878} C_VEL
LIN {X 0,Y 206.515,Z 861.039,A -85,B 0,C 180,E1 -20986.814,E2 -20986.814} C_VEL
LIN {X 0,Y 208.511,Z 856.375,A -85,B 0,C 180,E1 -20990.726,E2 -20990.726} C_VEL
LIN {X 0,Y 211.331,Z 850.611,A -85,B 0,C 180,E1 -20994.563,E2 -20994.563} C_VEL
LIN {X 0,Y 214.882,Z 843.658,A -85,B 0,C 180,E1 -20998.308,E2 -20998.308} C_VEL
LIN {X 0,Y 220.014,Z 834.179,A -85,B 0,C 180,E1 -21002.347,E2 -21002.347} C_VEL
LIN {X 0,Y 224.324,Z 826.038,A -85,B 0,C 180,E1 -21005.175,E2 -21005.175} C_VEL
LIN {X 0,Y 229.027,Z 816.835,A -85,B 0,C 180,E1 -21007.858,E2 -21007.858} C_VEL
LIN {X 0,Y 233.877,Z 807.049,A -85,B 0,C 180,E1 -21010.245,E2 -21010.245} C_VEL
LIN {X 0,Y 238.756,Z 796.834,A -85,B 0,C 180,E1 -21012.325,E2 -21012.325} C_VEL
LIN {X 0,Y 243.347,Z 786.27,A -85,B 0,C 180,E1 -21014.165,E2 -21014.165} C_VEL
LIN {X 0,Y 247.749,Z 775.464,A -85,B 0,C 180,E1 -21015.747,E2 -21015.747} C_VEL
LIN {X 0,Y 251.829,Z 764.53,A -85,B 0,C 180,E1 -21017.102,E2 -21017.102} C_VEL
LIN {X 0,Y 256.012,Z 752.052,A -85,B 0,C 180,E1 -21018.392,E2 -21018.392} C_VEL
LIN {X 0,Y 259.293,Z 740.893,A -85,B 0,C 180,E1 -21019.368,E2 -21019.368} C_VEL
LIN {X 0,Y 262.538,Z 728.395,A -85,B 0,C 180,E1 -21020.258,E2 -21020.258} C_VEL
LIN {X 0,Y 265.496,Z 714.693,A -85,B 0,C 180,E1 -21021.039,E2 -21021.039} C_VEL
LIN {X 0,Y 267.818,Z 701.327,A -85,B 0,C 180,E1 -21021.624,E2 -21021.624} C_VEL
LIN {X 0,Y 269.51,Z 687.875,A -85,B 0,C 180,E1 -21022.074,E2 -21022.074} C_VEL
LIN {X 0,Y 272.038,Z 654.171,A -85,B 0,C 180,E1 -21022.904,E2 -21022.904} C_VEL
LIN {X 0,Y 277.134,Z 581.193,A -85,B 0,C 180,E1 -21024.612,E2 -21024.612} C_VEL
LIN {X 0,Y 276.904,Z 579.991,A -85,B 0,C 180,E1 -21024.731,E2 -21024.731} C_VEL
LIN {X 0,Y 271.084,Z 566.498,A -85,B 0,C 180,E1 -21027.131,E2 -21027.131} C_VEL
LIN {X 0,Y 265.73,Z 555.615,A -85,B 0,C 180,E1 -21029.508,E2 -21029.508} C_VEL
LIN {X 0,Y 260.957,Z 546.603,A -85,B 0,C 180,E1 -21031.829,E2 -21031.829} C_VEL
LIN {X 0,Y 258.036,Z 541.681,A -85,B 0,C 180,E1 -21033.349,E2 -21033.349} C_VEL
LIN {X 0,Y 253.843,Z 535.691,A -85,B 0,C 180,E1 -21035.68,E2 -21035.68} C_VEL
LIN {X 0,Y 251.035,Z 531.808,A -85,B 0,C 180,E1 -21037.403,E2 -21037.403} C_VEL
LIN {X 0,Y 247.717,Z 527.416,A -85,B 0,C 180,E1 -21039.656,E2 -21039.656} C_VEL
LIN {X 0,Y 244.742,Z 523.424,A -85,B 0,C 180,E1 -21041.965,E2 -21041.965} C_VEL
LIN {X 0,Y 243.91,Z 522.466,A -85,B 0,C 180,E1 -21042.66,E2 -21042.66} C_VEL
LIN {X 0,Y 241.369,Z 519.343,A -85,B 0,C 180,E1 -21045.024,E2 -21045.024} C_VEL
LIN {X 0,Y 240.643,Z 517.91,A -85,B 0,C 180,E1 -21045.842,E2 -21045.842} C_VEL
LIN {X 0,Y 237.924,Z 515.474,A -85,B 0,C 180,E1 -21049.038,E2 -21049.038} C_VEL
LIN {X 0,Y 236.535,Z 512.509,A -85,B 0,C 180,E1 -21051.456,E2 -21051.456} C_VEL
LIN {X 0,Y 234.028,Z 510.515,A -85,B 0,C 180,E1 -21060,E2 -21060} C_VEL
LIN {X 0,Y 236.518,Z 512.492,A -85,B 0,C 180,E1 -21068.929,E2 -21068.929} C_VEL
LIN {X 0,Y 238.157,Z 515.789,A -85,B 0,C 180,E1 -21071.705,E2 -21071.705} C_VEL
LIN {X 0,Y 240.781,Z 518.261,A -85,B 0,C 180,E1 -21074.743,E2 -21074.743} C_VEL
LIN {X 0,Y 243.272,Z 521.95,A -85,B 0,C 180,E1 -21077.224,E2 -21077.224} C_VEL
LIN {X 0,Y 244.693,Z 523.44,A -85,B 0,C 180,E1 -21078.417,E2 -21078.417} C_VEL
LIN {X 0,Y 247.538,Z 527.287,A -85,B 0,C 180,E1 -21080.639,E2 -21080.639} C_VEL
LIN {X 0,Y 248.828,Z 528.82,A -85,B 0,C 180,E1 -21081.541,E2 -21081.541} C_VEL
LIN {X 0,Y 252.32,Z 533.576,A -85,B 0,C 180,E1 -21083.82,E2 -21083.82} C_VEL
LIN {X 0,Y 256.016,Z 538.79,A -85,B 0,C 180,E1 -21085.978,E2 -21085.978} C_VEL
LIN {X 0,Y 260.621,Z 545.406,A -85,B 0,C 180,E1 -21088.382,E2 -21088.382} C_VEL
LIN {X 0,Y 270.868,Z 560.022,A -85,B 0,C 180,E1 -21092.904,E2 -21092.904} C_VEL
LIN {X 0,Y 277.458,Z 567.497,A -85,B 0,C 180,E1 -21095.298,E2 -21095.298} C_VEL
LIN {X 0,Y 285.054,Z 574.867,A -85,B 0,C 180,E1 -21097.716,E2 -21097.716} C_VEL
LIN {X 0,Y 293.72,Z 582.251,A -85,B 0,C 180,E1 -21100.243,E2 -21100.243} C_VEL
LIN {X 0,Y 301.27,Z 588.639,A -85,B 0,C 180,E1 -21102.571,E2 -21102.571} C_VEL
LIN {X 0,Y 307.987,Z 594.607,A -85,B 0,C 180,E1 -21104.89,E2 -21104.89} C_VEL
LIN {X 0,Y 312.614,Z 598.651,A -85,B 0,C 180,E1 -21106.577,E2 -21106.577} C_VEL
LIN {X 0,Y 318.293,Z 603.641,A -85,B 0,C 180,E1 -21108.847,E2 -21108.847} C_VEL
LIN {X 0,Y 324.384,Z 609.314,A -85,B 0,C 180,E1 -21111.411,E2 -21111.411} C_VEL
LIN {X 0,Y 328.086,Z 612.494,A -85,B 0,C 180,E1 -21113.005,E2 -21113.005} C_VEL
LIN {X 0,Y 333.269,Z 616.977,A -85,B 0,C 180,E1 -21115.328,E2 -21115.328} C_VEL
LIN {X 0,Y 336.741,Z 619.887,A -85,B 0,C 180,E1 -21116.955,E2 -21116.955} C_VEL
LIN {X 0,Y 340.901,Z 623.536,A -85,B 0,C 180,E1 -21118.977,E2 -21118.977} C_VEL
LIN {X 0,Y 344.466,Z 626.36,A -85,B 0,C 180,E1 -21120.798,E2 -21120.798} C_VEL
LIN {X 0,Y 348.834,Z 630.412,A -85,B 0,C 180,E1 -21123.183,E2 -21123.183} C_VEL
LIN {X 0,Y 353.569,Z 633.773,A -85,B 0,C 180,E1 -21125.929,E2 -21125.929} C_VEL
LIN {X 0,Y 357.086,Z 637.113,A -85,B 0,C 180,E1 -21128.25,E2 -21128.25} C_VEL
LIN {X 0,Y 360.767,Z 639.737,A -85,B 0,C 180,E1 -21130.847,E2 -21130.847} C_VEL
LIN {X 0,Y 363.159,Z 641.22,A -85,B 0,C 180,E1 -21132.705,E2 -21132.705} C_VEL
LIN {X 0,Y 365.864,Z 644.013,A -85,B 0,C 180,E1 -21135.166,E2 -21135.166} C_VEL
LIN {X 0,Y 368.232,Z 645.944,A -85,B 0,C 180,E1 -21137.679,E2 -21137.679} C_VEL
LIN {X 0,Y 370.244,Z 647.057,A -85,B 0,C 180,E1 -21140.164,E2 -21140.164} C_VEL
LIN {X 0,Y 371.901,Z 647.876,A -85,B 0,C 180,E1 -21142.814,E2 -21142.814} C_VEL
LIN {X 0,Y 373.082,Z 648.561,A -85,B 0,C 180,E1 -21145.679,E2 -21145.679} C_VEL
LIN {X 0,Y 373.632,Z 648.721,A -85,B 0,C 180,E1 -21147.844,E2 -21147.844} C_VEL
LIN {X 0,Y 373.823,Z 648.856,A -85,B 0,C 180,E1 -21150,E2 -21150} C_VEL
LIN {X 0,Y 373.632,Z 648.721,A -85,B 0,C 180,E1 -21152.156,E2 -21152.156} C_VEL
LIN {X 0,Y 372.917,Z 648.484,A -85,B 0,C 180,E1 -21154.869,E2 -21154.869} C_VEL
LIN {X 0,Y 371.656,Z 647.73,A -85,B 0,C 180,E1 -21157.606,E2 -21157.606} C_VEL
LIN {X 0,Y 370.024,Z 647.052,A -85,B 0,C 180,E1 -21160.131,E2 -21160.131} C_VEL
LIN {X 0,Y 367.856,Z 645.678,A -85,B 0,C 180,E1 -21162.732,E2 -21162.732} C_VEL
LIN {X 0,Y 365.297,Z 643.475,A -85,B 0,C 180,E1 -21165.377,E2 -21165.377} C_VEL
LIN {X 0,Y 362.423,Z 640.625,A -85,B 0,C 180,E1 -21167.909,E2 -21167.909} C_VEL
LIN {X 0,Y 359.228,Z 638.686,A -85,B 0,C 180,E1 -21170.271,E2 -21170.271} C_VEL
LIN {X 0,Y 355.52,Z 635.768,A -85,B 0,C 180,E1 -21172.806,E2 -21172.806} C_VEL
LIN {X 0,Y 352.551,Z 632.941,A -85,B 0,C 180,E1 -21174.677,E2 -21174.677} C_VEL
LIN {X 0,Y 348.314,Z 629.991,A -85,B 0,C 180,E1 -21177.103,E2 -21177.103} C_VEL
LIN {X 0,Y 343.827,Z 625.704,A -85,B 0,C 180,E1 -21179.553,E2 -21179.553} C_VEL
LIN {X 0,Y 338.587,Z 621.635,A -85,B 0,C 180,E1 -21182.159,E2 -21182.159} C_VEL
LIN {X 0,Y 334.14,Z 617.661,A -85,B 0,C 180,E1 -21184.269,E2 -21184.269} C_VEL
LIN {X 0,Y 328.895,Z 613.261,A -85,B 0,C 180,E1 -21186.637,E2 -21186.637} C_VEL
LIN {X 0,Y 324.868,Z 609.647,A -85,B 0,C 180,E1 -21188.387,E2 -21188.387} C_VEL
LIN {X 0,Y 319.609,Z 604.919,A -85,B 0,C 180,E1 -21190.608,E2 -21190.608} C_VEL
LIN {X 0,Y 312.923,Z 598.967,A -85,B 0,C 180,E1 -21193.297,E2 -21193.297} C_VEL
LIN {X 0,Y 308.237,Z 594.79,A -85,B 0,C 180,E1 -21195.024,E2 -21195.024} C_VEL
LIN {X 0,Y 302.947,Z 589.982,A -85,B 0,C 180,E1 -21196.861,E2 -21196.861} C_VEL
LIN {X 0,Y 296.836,Z 584.852,A -85,B 0,C 180,E1 -21198.832,E2 -21198.832} C_VEL
LIN {X 0,Y 288.698,Z 578.02,A -85,B 0,C 180,E1 -21201.228,E2 -21201.228} C_VEL
LIN {X 0,Y 279.42,Z 569.531,A -85,B 0,C 180,E1 -21204.046,E2 -21204.046} C_VEL
LIN {X 0,Y 271.93,Z 561.294,A -85,B 0,C 180,E1 -21206.688,E2 -21206.688} C_VEL
LIN {X 0,Y 266.442,Z 554.093,A -85,B 0,C 180,E1 -21208.913,E2 -21208.913} C_VEL
LIN {X 0,Y 259.103,Z 543.247,A -85,B 0,C 180,E1 -21212.379,E2 -21212.379} C_VEL
LIN {X 0,Y 254.178,Z 536.119,A -85,B 0,C 180,E1 -21215.07,E2 -21215.07} C_VEL
LIN {X 0,Y 250.774,Z 531.429,A -85,B 0,C 180,E1 -21217.157,E2 -21217.157} C_VEL
LIN {X 0,Y 247.778,Z 527.483,A -85,B 0,C 180,E1 -21219.197,E2 -21219.197} C_VEL
LIN {X 0,Y 245.043,Z 524.042,A -85,B 0,C 180,E1 -21221.281,E2 -21221.281} C_VEL
LIN {X 0,Y 244.224,Z 522.8,A -85,B 0,C 180,E1 -21221.98,E2 -21221.98} C_VEL
LIN {X 0,Y 241.484,Z 519.592,A -85,B 0,C 180,E1 -21224.48,E2 -21224.48} C_VEL
LIN {X 0,Y 240.454,Z 517.808,A -85,B 0,C 180,E1 -21225.615,E2 -21225.615} C_VEL
LIN {X 0,Y 237.792,Z 515.271,A -85,B 0,C 180,E1 -21228.817,E2 -21228.817} C_VEL
LIN {X 0,Y 236.517,Z 512.496,A -85,B 0,C 180,E1 -21231.071,E2 -21231.071} C_VEL
LIN {X 0,Y 234.086,Z 510.693,A -85,B 0,C 180,E1 -21238.28,E2 -21238.28} C_VEL
LIN {X 0,Y 234.058,Z 510.591,A -85,B 0,C 180,E1 -21240.861,E2 -21240.861} C_VEL
LIN {X 0,Y 236.587,Z 512.643,A -85,B 0,C 180,E1 -21248.65,E2 -21248.65} C_VEL
LIN {X 0,Y 238.223,Z 515.87,A -85,B 0,C 180,E1 -21251.379,E2 -21251.379} C_VEL
LIN {X 0,Y 240.823,Z 518.24,A -85,B 0,C 180,E1 -21254.363,E2 -21254.363} C_VEL
LIN {X 0,Y 242.997,Z 521.594,A -85,B 0,C 180,E1 -21256.56,E2 -21256.56} C_VEL
LIN {X 0,Y 244.685,Z 523.323,A -85,B 0,C 180,E1 -21257.985,E2 -21257.985} C_VEL
LIN {X 0,Y 247.44,Z 527.143,A -85,B 0,C 180,E1 -21260.15,E2 -21260.15} C_VEL
LIN {X 0,Y 248.828,Z 528.874,A -85,B 0,C 180,E1 -21261.129,E2 -21261.129} C_VEL
LIN {X 0,Y 252.219,Z 533.421,A -85,B 0,C 180,E1 -21263.341,E2 -21263.341} C_VEL
LIN {X 0,Y 255.739,Z 538.407,A -85,B 0,C 180,E1 -21265.409,E2 -21265.409} C_VEL
LIN {X 0,Y 259.674,Z 544.194,A -85,B 0,C 180,E1 -21267.503,E2 -21267.503} C_VEL
LIN {X 0,Y 264.901,Z 554.036,A -85,B 0,C 180,E1 -21270.106,E2 -21270.106} C_VEL
LIN {X 0,Y 270.076,Z 564.334,A -85,B 0,C 180,E1 -21272.435,E2 -21272.435} C_VEL
LIN {X 0,Y 276.34,Z 578.5,A -85,B 0,C 180,E1 -21275.039,E2 -21275.039} C_VEL
LIN {X 0,Y 277.117,Z 580.406,A -85,B 0,C 180,E1 -21275.349,E2 -21275.349} C_VEL
LIN {X 0,Y 272.042,Z 654.172,A -85,B 0,C 180,E1 -21277.097,E2 -21277.097} C_VEL
LIN {X 0,Y 269.495,Z 687.889,A -85,B 0,C 180,E1 -21277.922,E2 -21277.922} C_VEL
LIN {X 0,Y 267.66,Z 702.326,A -85,B 0,C 180,E1 -21278.409,E2 -21278.409} C_VEL
LIN {X 0,Y 264.62,Z 719.233,A -85,B 0,C 180,E1 -21279.18,E2 -21279.18} C_VEL
LIN {X 0,Y 262.056,Z 730.422,A -85,B 0,C 180,E1 -21279.862,E2 -21279.862} C_VEL
LIN {X 0,Y 260.305,Z 735.949,A -85,B 0,C 180,E1 -21280.119,E2 -21280.119} C_VEL
LIN {X 0,Y 255.989,Z 744.838,A -85,B 0,C 180,E1 -21280.329,E2 -21280.329} C_VEL
LIN {X 0,Y 251.342,Z 753.479,A -85,B 0,C 180,E1 -21280.638,E2 -21280.638} C_VEL
LIN {X 0,Y 249.085,Z 758.615,A -85,B 0,C 180,E1 -21281.057,E2 -21281.057} C_VEL
LIN {X 0,Y 244.398,Z 771.34,A -85,B 0,C 180,E1 -21282.535,E2 -21282.535} C_VEL
LIN {X 0,Y 239.743,Z 782.628,A -85,B 0,C 180,E1 -21284.095,E2 -21284.095} C_VEL
LIN {X 0,Y 234.984,Z 793.361,A -85,B 0,C 180,E1 -21285.873,E2 -21285.873} C_VEL
LIN {X 0,Y 230.288,Z 803.289,A -85,B 0,C 180,E1 -21287.826,E2 -21287.826} C_VEL
LIN {X 0,Y 225.017,Z 813.49,A -85,B 0,C 180,E1 -21290.188,E2 -21290.188} C_VEL
LIN {X 0,Y 220.249,Z 822.447,A -85,B 0,C 180,E1 -21292.68,E2 -21292.68} C_VEL
LIN {X 0,Y 216.003,Z 830.341,A -85,B 0,C 180,E1 -21295.293,E2 -21295.293} C_VEL
LIN {X 0,Y 212.005,Z 837.302,A -85,B 0,C 180,E1 -21297.968,E2 -21297.968} C_VEL
LIN {X 0,Y 208.57,Z 843.444,A -85,B 0,C 180,E1 -21300.753,E2 -21300.753} C_VEL
LIN {X 0,Y 204.752,Z 850.396,A -85,B 0,C 180,E1 -21304.593,E2 -21304.593} C_VEL
LIN {X 0,Y 201.768,Z 856.162,A -85,B 0,C 180,E1 -21308.548,E2 -21308.548} C_VEL
LIN {X 0,Y 200.104,Z 859.784,A -85,B 0,C 180,E1 -21311.573,E2 -21311.573} C_VEL
LIN {X 0,Y 198.421,Z 863.644,A -85,B 0,C 180,E1 -21315.645,E2 -21315.645} C_VEL
LIN {X 0,Y 197.51,Z 866.508,A -85,B 0,C 180,E1 -21319.752,E2 -21319.752} C_VEL
LIN {X 0,Y 197.301,Z 867.651,A -85,B 0,C 180,E1 -21321.809,E2 -21321.809} C_VEL
LIN {X 0,Y 197.205,Z 869.162,A -85,B 0,C 180,E1 -21326.256,E2 -21326.256} C_VEL
LIN {X 0,Y 197.326,Z 869.571,A -85,B 0,C 180,E1 -21330,E2 -21330} C_VEL
LIN {X 0,Y 197.204,Z 869.09,A -85,B 0,C 180,E1 -21334.087,E2 -21334.087} C_VEL
LIN {X 0,Y 197.301,Z 867.651,A -85,B 0,C 180,E1 -21338.191,E2 -21338.191} C_VEL
LIN {X 0,Y 197.837,Z 865.25,A -85,B 0,C 180,E1 -21342.306,E2 -21342.306} C_VEL
LIN {X 0,Y 199.63,Z 860.826,A -85,B 0,C 180,E1 -21347.412,E2 -21347.412} C_VEL
LIN {X 0,Y 201.16,Z 857.451,A -85,B 0,C 180,E1 -21350.448,E2 -21350.448} C_VEL
LIN {X 0,Y 203.924,Z 851.942,A -85,B 0,C 180,E1 -21354.428,E2 -21354.428} C_VEL
LIN {X 0,Y 206.523,Z 847.118,A -85,B 0,C 180,E1 -21357.324,E2 -21357.324} C_VEL
LIN {X 0,Y 210.803,Z 839.408,A -85,B 0,C 180,E1 -21361.114,E2 -21361.114} C_VEL
LIN {X 0,Y 214.629,Z 832.757,A -85,B 0,C 180,E1 -21363.824,E2 -21363.824} C_VEL
LIN {X 0,Y 219.191,Z 824.392,A -85,B 0,C 180,E1 -21366.718,E2 -21366.718} C_VEL
LIN {X 0,Y 223.372,Z 816.622,A -85,B 0,C 180,E1 -21368.995,E2 -21368.995} C_VEL
LIN {X 0,Y 228.431,Z 806.836,A -85,B 0,C 180,E1 -21371.411,E2 -21371.411} C_VEL
LIN {X 0,Y 233.499,Z 796.622,A -85,B 0,C 180,E1 -21373.511,E2 -21373.511} C_VEL
LIN {X 0,Y 238.763,Z 784.916,A -85,B 0,C 180,E1 -21375.544,E2 -21375.544} C_VEL
LIN {X 0,Y 243.305,Z 773.947,A -85,B 0,C 180,E1 -21377.135,E2 -21377.135} C_VEL
LIN {X 0,Y 247.544,Z 762.819,A -85,B 0,C 180,E1 -21378.486,E2 -21378.486} C_VEL
LIN {X 0,Y 251.254,Z 752.08,A -85,B 0,C 180,E1 -21379.586,E2 -21379.586} C_VEL
LIN {X 0,Y 255.157,Z 739.022,A -85,B 0,C 180,E1 -21380.714,E2 -21380.714} C_VEL
LIN {X 0,Y 258.35,Z 726.826,A -85,B 0,C 180,E1 -21381.561,E2 -21381.561} C_VEL
LIN {X 0,Y 261.248,Z 713.718,A -85,B 0,C 180,E1 -21382.285,E2 -21382.285} C_VEL
LIN {X 0,Y 263.469,Z 701.117,A -85,B 0,C 180,E1 -21382.834,E2 -21382.834} C_VEL
LIN {X 0,Y 265.215,Z 687.665,A -85,B 0,C 180,E1 -21383.282,E2 -21383.282} C_VEL
LIN {X 0,Y 267.561,Z 657.544,A -85,B 0,C 180,E1 -21384.031,E2 -21384.031} C_VEL
LIN {X 0,Y 272.892,Z 583.458,A -85,B 0,C 180,E1 -21385.772,E2 -21385.772} C_VEL
LIN {X 0,Y 267.843,Z 571.441,A -85,B 0,C 180,E1 -21387.967,E2 -21387.967} C_VEL
LIN {X 0,Y 262.499,Z 560.336,A -85,B 0,C 180,E1 -21390.461,E2 -21390.461} C_VEL
LIN {X 0,Y 258.295,Z 552.176,A -85,B 0,C 180,E1 -21392.612,E2 -21392.612} C_VEL
LIN {X 0,Y 255.545,Z 547.404,A -85,B 0,C 180,E1 -21394.113,E2 -21394.113} C_VEL
LIN {X 0,Y 251.549,Z 541.644,A -85,B 0,C 180,E1 -21396.434,E2 -21396.434} C_VEL
LIN {X 0,Y 249.193,Z 538.245,A -85,B 0,C 180,E1 -21397.948,E2 -21397.948} C_VEL
LIN {X 0,Y 246.038,Z 533.97,A -85,B 0,C 180,E1 -21400.171,E2 -21400.171} C_VEL
LIN {X 0,Y 243.158,Z 529.989,A -85,B 0,C 180,E1 -21402.498,E2 -21402.498} C_VEL
LIN {X 0,Y 239.914,Z 525.887,A -85,B 0,C 180,E1 -21405.582,E2 -21405.582} C_VEL
LIN {X 0,Y 239.196,Z 524.664,A -85,B 0,C 180,E1 -21406.405,E2 -21406.405} C_VEL
LIN {X 0,Y 236.562,Z 521.982,A -85,B 0,C 180,E1 -21409.732,E2 -21409.732} C_VEL
LIN {X 0,Y 235.434,Z 519.422,A -85,B 0,C 180,E1 -21411.848,E2 -21411.848} C_VEL
LIN {X 0,Y 233.162,Z 517.564,A -85,B 0,C 180,E1 -21420,E2 -21420} C_VEL
LIN {X 0,Y 235.489,Z 519.517,A -85,B 0,C 180,E1 -21428.678,E2 -21428.678} C_VEL
LIN {X 0,Y 237.027,Z 522.669,A -85,B 0,C 180,E1 -21431.382,E2 -21431.382} C_VEL
LIN {X 0,Y 239.441,Z 525.011,A -85,B 0,C 180,E1 -21434.289,E2 -21434.289} C_VEL
LIN {X 0,Y 241.962,Z 528.772,A -85,B 0,C 180,E1 -21436.885,E2 -21436.885} C_VEL
LIN {X 0,Y 243.276,Z 530.275,A -85,B 0,C 180,E1 -21438.031,E2 -21438.031} C_VEL
LIN {X 0,Y 246.193,Z 534.16,A -85,B 0,C 180,E1 -21440.359,E2 -21440.359} C_VEL
LIN {X 0,Y 250.243,Z 539.683,A -85,B 0,C 180,E1 -21443.152,E2 -21443.152} C_VEL
LIN {X 0,Y 255.583,Z 547.416,A -85,B 0,C 180,E1 -21446.321,E2 -21446.321} C_VEL
LIN {X 0,Y 260.964,Z 555.781,A -85,B 0,C 180,E1 -21449.106,E2 -21449.106} C_VEL
LIN {X 0,Y 268.768,Z 566.644,A -85,B 0,C 180,E1 -21452.526,E2 -21452.526} C_VEL
LIN {X 0,Y 275.063,Z 573.837,A -85,B 0,C 180,E1 -21454.868,E2 -21454.868} C_VEL
LIN {X 0,Y 282.571,Z 581.22,A -85,B 0,C 180,E1 -21457.318,E2 -21457.318} C_VEL
LIN {X 0,Y 292.107,Z 589.253,A -85,B 0,C 180,E1 -21460.098,E2 -21460.098} C_VEL
LIN {X 0,Y 298.562,Z 594.78,A -85,B 0,C 180,E1 -21462.083,E2 -21462.083} C_VEL
LIN {X 0,Y 303.239,Z 598.771,A -85,B 0,C 180,E1 -21463.613,E2 -21463.613} C_VEL
LIN {X 0,Y 309.914,Z 604.497,A -85,B 0,C 180,E1 -21465.955,E2 -21465.955} C_VEL
LIN {X 0,Y 315.507,Z 609.493,A -85,B 0,C 180,E1 -21468.128,E2 -21468.128} C_VEL
LIN {X 0,Y 322.565,Z 615.881,A -85,B 0,C 180,E1 -21471.052,E2 -21471.052} C_VEL
LIN {X 0,Y 326.714,Z 619.459,A -85,B 0,C 180,E1 -21472.835,E2 -21472.835} C_VEL
LIN {X 0,Y 331.865,Z 623.845,A -85,B 0,C 180,E1 -21475.126,E2 -21475.126} C_VEL
LIN {X 0,Y 335.277,Z 626.697,A -85,B 0,C 180,E1 -21476.708,E2 -21476.708} C_VEL
LIN {X 0,Y 339.853,Z 630.639,A -85,B 0,C 180,E1 -21478.928,E2 -21478.928} C_VEL
LIN {X 0,Y 343.207,Z 633.323,A -85,B 0,C 180,E1 -21480.627,E2 -21480.627} C_VEL
LIN {X 0,Y 347.751,Z 637.43,A -85,B 0,C 180,E1 -21483.093,E2 -21483.093} C_VEL
LIN {X 0,Y 352.452,Z 640.783,A -85,B 0,C 180,E1 -21485.81,E2 -21485.81} C_VEL
LIN {X 0,Y 355.972,Z 644.056,A -85,B 0,C 180,E1 -21488.112,E2 -21488.112} C_VEL
LIN {X 0,Y 359.806,Z 646.769,A -85,B 0,C 180,E1 -21490.794,E2 -21490.794} C_VEL
LIN {X 0,Y 362.112,Z 648.195,A -85,B 0,C 180,E1 -21492.578,E2 -21492.578} C_VEL
LIN {X 0,Y 364.751,Z 650.914,A -85,B 0,C 180,E1 -21494.947,E2 -21494.947} C_VEL
LIN {X 0,Y 367.165,Z 652.858,A -85,B 0,C 180,E1 -21497.473,E2 -21497.473} C_VEL
LIN {X 0,Y 368.978,Z 653.947,A -85,B 0,C 180,E1 -21499.621,E2 -21499.621} C_VEL
LIN {X 0,Y 370.774,Z 654.776,A -85,B 0,C 180,E1 -21502.375,E2 -21502.375} C_VEL
LIN {X 0,Y 372.048,Z 655.523,A -85,B 0,C 180,E1 -21505.119,E2 -21505.119} C_VEL
LIN {X 0,Y 372.765,Z 655.755,A -85,B 0,C 180,E1 -21507.839,E2 -21507.839} C_VEL
LIN {X 0,Y 372.958,Z 655.902,A -85,B 0,C 180,E1 -21510,E2 -21510} C_VEL
LIN {X 0,Y 372.755,Z 655.747,A -85,B 0,C 180,E1 -21512.204,E2 -21512.204} C_VEL
LIN {X 0,Y 372.048,Z 655.528,A -85,B 0,C 180,E1 -21514.881,E2 -21514.881} C_VEL
LIN {X 0,Y 370.774,Z 654.776,A -85,B 0,C 180,E1 -21517.625,E2 -21517.625} C_VEL
LIN {X 0,Y 369.066,Z 654.036,A -85,B 0,C 180,E1 -21520.262,E2 -21520.262} C_VEL
LIN {X 0,Y 366.801,Z 652.608,A -85,B 0,C 180,E1 -21522.935,E2 -21522.935} C_VEL
LIN {X 0,Y 364.255,Z 650.452,A -85,B 0,C 180,E1 -21525.509,E2 -21525.509} C_VEL
LIN {X 0,Y 361.256,Z 647.508,A -85,B 0,C 180,E1 -21528.135,E2 -21528.135} C_VEL
LIN {X 0,Y 358.032,Z 645.577,A -85,B 0,C 180,E1 -21530.478,E2 -21530.478} C_VEL
LIN {X 0,Y 354.264,Z 642.63,A -85,B 0,C 180,E1 -21533.019,E2 -21533.019} C_VEL
LIN {X 0,Y 351.366,Z 639.872,A -85,B 0,C 180,E1 -21534.837,E2 -21534.837} C_VEL
LIN {X 0,Y 347.09,Z 636.911,A -85,B 0,C 180,E1 -21537.265,E2 -21537.265} C_VEL
LIN {X 0,Y 342.396,Z 632.507,A -85,B 0,C 180,E1 -21539.8,E2 -21539.8} C_VEL
LIN {X 0,Y 337.065,Z 628.396,A -85,B 0,C 180,E1 -21542.428,E2 -21542.428} C_VEL
LIN {X 0,Y 332.547,Z 624.354,A -85,B 0,C 180,E1 -21544.564,E2 -21544.564} C_VEL
LIN {X 0,Y 327.137,Z 619.854,A -85,B 0,C 180,E1 -21546.979,E2 -21546.979} C_VEL
LIN {X 0,Y 322.889,Z 616.097,A -85,B 0,C 180,E1 -21548.811,E2 -21548.811} C_VEL
LIN {X 0,Y 317.516,Z 611.243,A -85,B 0,C 180,E1 -21551.057,E2 -21551.057} C_VEL
LIN {X 0,Y 311.072,Z 605.633,A -85,B 0,C 180,E1 -21553.602,E2 -21553.602} C_VEL
LIN {X 0,Y 306.564,Z 601.598,A -85,B 0,C 180,E1 -21555.243,E2 -21555.243} C_VEL
LIN {X 0,Y 300.061,Z 595.922,A -85,B 0,C 180,E1 -21557.458,E2 -21557.458} C_VEL
LIN {X 0,Y 294.03,Z 590.869,A -85,B 0,C 180,E1 -21559.323,E2 -21559.323} C_VEL
LIN {X 0,Y 286.096,Z 584.311,A -85,B 0,C 180,E1 -21561.636,E2 -21561.636} C_VEL
LIN {X 0,Y 276.653,Z 575.535,A -85,B 0,C 180,E1 -21564.584,E2 -21564.584} C_VEL
LIN {X 0,Y 269.238,Z 567.221,A -85,B 0,C 180,E1 -21567.288,E2 -21567.288} C_VEL
LIN {X 0,Y 261.817,Z 557.116,A -85,B 0,C 180,E1 -21570.484,E2 -21570.484} C_VEL
LIN {X 0,Y 256.437,Z 548.772,A -85,B 0,C 180,E1 -21573.209,E2 -21573.209} C_VEL
LIN {X 0,Y 251.704,Z 541.818,A -85,B 0,C 180,E1 -21575.926,E2 -21575.926} C_VEL
LIN {X 0,Y 248.775,Z 537.694,A -85,B 0,C 180,E1 -21577.81,E2 -21577.81} C_VEL
LIN {X 0,Y 245.927,Z 533.858,A -85,B 0,C 180,E1 -21579.836,E2 -21579.836} C_VEL
LIN {X 0,Y 243.276,Z 530.276,A -85,B 0,C 180,E1 -21581.969,E2 -21581.969} C_VEL
LIN {X 0,Y 241.962,Z 528.772,A -85,B 0,C 180,E1 -21583.115,E2 -21583.115} C_VEL
LIN {X 0,Y 239.571,Z 525.273,A -85,B 0,C 180,E1 -21585.556,E2 -21585.556} C_VEL
LIN {X 0,Y 238.827,Z 524.429,A -85,B 0,C 180,E1 -21586.384,E2 -21586.384} C_VEL
LIN {X 0,Y 236.44,Z 521.777,A -85,B 0,C 180,E1 -21589.511,E2 -21589.511} C_VEL
LIN {X 0,Y 235.443,Z 519.426,A -85,B 0,C 180,E1 -21591.417,E2 -21591.417} C_VEL
LIN {X 0,Y 233.162,Z 517.566,A -85,B 0,C 180,E1 -21600,E2 -21600} C_VEL
LIN {X 0,Y 235.493,Z 519.464,A -85,B 0,C 180,E1 -21608.258,E2 -21608.258} C_VEL
LIN {X 0,Y 236.944,Z 522.552,A -85,B 0,C 180,E1 -21610.846,E2 -21610.846} C_VEL
LIN {X 0,Y 239.562,Z 525.164,A -85,B 0,C 180,E1 -21614.007,E2 -21614.007} C_VEL
LIN {X 0,Y 241.781,Z 528.515,A -85,B 0,C 180,E1 -21616.299,E2 -21616.299} C_VEL
LIN {X 0,Y 243.24,Z 530.12,A -85,B 0,C 180,E1 -21617.574,E2 -21617.574} C_VEL
LIN {X 0,Y 246.036,Z 533.986,A -85,B 0,C 180,E1 -21619.829,E2 -21619.829} C_VEL
LIN {X 0,Y 250.213,Z 539.665,A -85,B 0,C 180,E1 -21622.719,E2 -21622.719} C_VEL
LIN {X 0,Y 253.507,Z 544.455,A -85,B 0,C 180,E1 -21624.737,E2 -21624.737} C_VEL
LIN {X 0,Y 257.212,Z 550.101,A -85,B 0,C 180,E1 -21626.798,E2 -21626.798} C_VEL
LIN {X 0,Y 261.854,Z 559.015,A -85,B 0,C 180,E1 -21629.219,E2 -21629.219} C_VEL
LIN {X 0,Y 266.91,Z 569.387,A -85,B 0,C 180,E1 -21631.611,E2 -21631.611} C_VEL
LIN {X 0,Y 272.836,Z 583.198,A -85,B 0,C 180,E1 -21634.199,E2 -21634.199} C_VEL
LIN {X 0,Y 268.618,Z 642.923,A -85,B 0,C 180,E1 -21635.628,E2 -21635.628} C_VEL
LIN {X 0,Y 265.351,Z 686.344,A -85,B 0,C 180,E1 -21636.679,E2 -21636.679} C_VEL
LIN {X 0,Y 263.596,Z 700.117,A -85,B 0,C 180,E1 -21637.123,E2 -21637.123} C_VEL
LIN {X 0,Y 261.359,Z 712.95,A -85,B 0,C 180,E1 -21637.668,E2 -21637.668} C_VEL
LIN {X 0,Y 258.636,Z 725.467,A -85,B 0,C 180,E1 -21638.347,E2 -21638.347} C_VEL
LIN {X 0,Y 255.601,Z 737.358,A -85,B 0,C 180,E1 -21639.155,E2 -21639.155} C_VEL
LIN {X 0,Y 252.212,Z 748.996,A -85,B 0,C 180,E1 -21640.123,E2 -21640.123} C_VEL
LIN {X 0,Y 249.085,Z 758.615,A -85,B 0,C 180,E1 -21641.057,E2 -21641.057} C_VEL
LIN {X 0,Y 246.751,Z 763.821,A -85,B 0,C 180,E1 -21641.508,E2 -21641.508} C_VEL
LIN {X 0,Y 236.308,Z 780.093,A -85,B 0,C 180,E1 -21642.587,E2 -21642.587} C_VEL
LIN {X 0,Y 233.812,Z 784.658,A -85,B 0,C 180,E1 -21643.193,E2 -21643.193} C_VEL
LIN {X 0,Y 229.559,Z 793.846,A -85,B 0,C 180,E1 -21644.761,E2 -21644.761} C_VEL
LIN {X 0,Y 225.024,Z 803.077,A -85,B 0,C 180,E1 -21646.6,E2 -21646.6} C_VEL
LIN {X 0,Y 219.542,Z 813.278,A -85,B 0,C 180,E1 -21648.987,E2 -21648.987} C_VEL
LIN {X 0,Y 214.558,Z 822.234,A -85,B 0,C 180,E1 -21651.512,E2 -21651.512} C_VEL
LIN {X 0,Y 210.082,Z 830.126,A -85,B 0,C 180,E1 -21654.167,E2 -21654.167} C_VEL
LIN {X 0,Y 205.928,Z 837.089,A -85,B 0,C 180,E1 -21656.904,E2 -21656.904} C_VEL
LIN {X 0,Y 202.292,Z 843.23,A -85,B 0,C 180,E1 -21659.752,E2 -21659.752} C_VEL
LIN {X 0,Y 198.242,Z 850.182,A -85,B 0,C 180,E1 -21663.696,E2 -21663.696} C_VEL
LIN {X 0,Y 195.062,Z 855.948,A -85,B 0,C 180,E1 -21667.771,E2 -21667.771} C_VEL
LIN {X 0,Y 193.204,Z 859.717,A -85,B 0,C 180,E1 -21671.045,E2 -21671.045} C_VEL
LIN {X 0,Y 191.48,Z 863.432,A -85,B 0,C 180,E1 -21675.113,E2 -21675.113} C_VEL
LIN {X 0,Y 190.45,Z 866.296,A -85,B 0,C 180,E1 -21679.368,E2 -21679.368} C_VEL
LIN {X 0,Y 190.219,Z 867.44,A -85,B 0,C 180,E1 -21681.501,E2 -21681.501} C_VEL
LIN {X 0,Y 190.123,Z 868.988,A -85,B 0,C 180,E1 -21686.44,E2 -21686.44} C_VEL
LIN {X 0,Y 190.231,Z 869.362,A -85,B 0,C 180,E1 -21690,E2 -21690} C_VEL
LIN {X 0,Y 190.123,Z 868.88,A -85,B 0,C 180,E1 -21694.24,E2 -21694.24} C_VEL
LIN {X 0,Y 190.219,Z 867.44,A -85,B 0,C 180,E1 -21698.499,E2 -21698.499} C_VEL
LIN {X 0,Y 190.826,Z 865.038,A -85,B 0,C 180,E1 -21702.766,E2 -21702.766} C_VEL
LIN {X 0,Y 192.298,Z 861.655,A -85,B 0,C 180,E1 -21707,E2 -21707} C_VEL
LIN {X 0,Y 194.427,Z 857.238,A -85,B 0,C 180,E1 -21711.19,E2 -21711.19} C_VEL
LIN {X 0,Y 197.378,Z 851.729,A -85,B 0,C 180,E1 -21715.295,E2 -21715.295} C_VEL
LIN {X 0,Y 199.988,Z 847.163,A -85,B 0,C 180,E1 -21718.133,E2 -21718.133} C_VEL
LIN {X 0,Y 204.637,Z 839.194,A -85,B 0,C 180,E1 -21722.162,E2 -21722.162} C_VEL
LIN {X 0,Y 208.696,Z 832.545,A -85,B 0,C 180,E1 -21724.923,E2 -21724.923} C_VEL
LIN {X 0,Y 213.051,Z 824.881,A -85,B 0,C 180,E1 -21727.655,E2 -21727.655} C_VEL
LIN {X 0,Y 217.812,Z 816.408,A -85,B 0,C 180,E1 -21730.189,E2 -21730.189} C_VEL
LIN {X 0,Y 223.073,Z 806.623,A -85,B 0,C 180,E1 -21732.637,E2 -21732.637} C_VEL
LIN {X 0,Y 228.813,Z 795.403,A -85,B 0,C 180,E1 -21734.945,E2 -21734.945} C_VEL
LIN {X 0,Y 233.793,Z 784.703,A -85,B 0,C 180,E1 -21736.799,E2 -21736.799} C_VEL
LIN {X 0,Y 238.499,Z 773.736,A -85,B 0,C 180,E1 -21738.393,E2 -21738.393} C_VEL
LIN {X 0,Y 242.881,Z 762.609,A -85,B 0,C 180,E1 -21739.744,E2 -21739.744} C_VEL
LIN {X 0,Y 247.047,Z 750.712,A -85,B 0,C 180,E1 -21740.96,E2 -21740.96} C_VEL
LIN {X 0,Y 250.817,Z 738.42,A -85,B 0,C 180,E1 -21742.004,E2 -21742.004} C_VEL
LIN {X 0,Y 254.076,Z 726.246,A -85,B 0,C 180,E1 -21742.841,E2 -21742.841} C_VEL
LIN {X 0,Y 256.944,Z 713.507,A -85,B 0,C 180,E1 -21743.543,E2 -21743.543} C_VEL
LIN {X 0,Y 259.245,Z 700.908,A -85,B 0,C 180,E1 -21744.084,E2 -21744.084} C_VEL
LIN {X 0,Y 261.025,Z 687.455,A -85,B 0,C 180,E1 -21744.533,E2 -21744.533} C_VEL
LIN {X 0,Y 263.708,Z 653.751,A -85,B 0,C 180,E1 -21745.368,E2 -21745.368} C_VEL
LIN {X 0,Y 268.719,Z 586.238,A -85,B 0,C 180,E1 -21746.959,E2 -21746.959} C_VEL
LIN {X 0,Y 264.019,Z 574.986,A -85,B 0,C 180,E1 -21749.124,E2 -21749.124} C_VEL
LIN {X 0,Y 258.39,Z 562.959,A -85,B 0,C 180,E1 -21751.945,E2 -21751.945} C_VEL
LIN {X 0,Y 254.24,Z 555.03,A -85,B 0,C 180,E1 -21754.234,E2 -21754.234} C_VEL
LIN {X 0,Y 249.919,Z 548.381,A -85,B 0,C 180,E1 -21756.815,E2 -21756.815} C_VEL
LIN {X 0,Y 246.891,Z 544.056,A -85,B 0,C 180,E1 -21758.832,E2 -21758.832} C_VEL
LIN {X 0,Y 244.386,Z 540.542,A -85,B 0,C 180,E1 -21760.688,E2 -21760.688} C_VEL
LIN {X 0,Y 241.096,Z 535.955,A -85,B 0,C 180,E1 -21763.488,E2 -21763.488} C_VEL
LIN {X 0,Y 238.482,Z 532.43,A -85,B 0,C 180,E1 -21766.146,E2 -21766.146} C_VEL
LIN {X 0,Y 237.964,Z 531.516,A -85,B 0,C 180,E1 -21766.768,E2 -21766.768} C_VEL
LIN {X 0,Y 235.425,Z 528.794,A -85,B 0,C 180,E1 -21770.115,E2 -21770.115} C_VEL
LIN {X 0,Y 234.339,Z 526.379,A -85,B 0,C 180,E1 -21772.243,E2 -21772.243} C_VEL
LIN {X 0,Y 232.299,Z 524.591,A -85,B 0,C 180,E1 -21780,E2 -21780} C_VEL
LIN {X 0,Y 234.442,Z 526.471,A -85,B 0,C 180,E1 -21788.371,E2 -21788.371} C_VEL
LIN {X 0,Y 235.976,Z 529.647,A -85,B 0,C 180,E1 -21791.162,E2 -21791.162} C_VEL
LIN {X 0,Y 238.236,Z 531.985,A -85,B 0,C 180,E1 -21793.977,E2 -21793.977} C_VEL
LIN {X 0,Y 240.771,Z 535.706,A -85,B 0,C 180,E1 -21796.643,E2 -21796.643} C_VEL
LIN {X 0,Y 241.859,Z 537.06,A -85,B 0,C 180,E1 -21797.628,E2 -21797.628} C_VEL
LIN {X 0,Y 244.804,Z 541.004,A -85,B 0,C 180,E1 -21800.042,E2 -21800.042} C_VEL
LIN {X 0,Y 248.548,Z 546.42,A -85,B 0,C 180,E1 -21802.714,E2 -21802.714} C_VEL
LIN {X 0,Y 253.351,Z 553.506,A -85,B 0,C 180,E1 -21805.667,E2 -21805.667} C_VEL
LIN {X 0,Y 258.424,Z 561.603,A -85,B 0,C 180,E1 -21808.406,E2 -21808.406} C_VEL
LIN {X 0,Y 265.96,Z 572.378,A -85,B 0,C 180,E1 -21811.847,E2 -21811.847} C_VEL
LIN {X 0,Y 272.502,Z 580.031,A -85,B 0,C 180,E1 -21814.367,E2 -21814.367} C_VEL
LIN {X 0,Y 280.181,Z 587.637,A -85,B 0,C 180,E1 -21816.937,E2 -21816.937} C_VEL
LIN {X 0,Y 289.811,Z 595.744,A -85,B 0,C 180,E1 -21819.757,E2 -21819.757} C_VEL
LIN {X 0,Y 296.749,Z 601.558,A -85,B 0,C 180,E1 -21821.86,E2 -21821.86} C_VEL
LIN {X 0,Y 304.005,Z 607.742,A -85,B 0,C 180,E1 -21824.222,E2 -21824.222} C_VEL
LIN {X 0,Y 310.387,Z 613.322,A -85,B 0,C 180,E1 -21826.531,E2 -21826.531} C_VEL
LIN {X 0,Y 316.488,Z 618.62,A -85,B 0,C 180,E1 -21828.937,E2 -21828.937} C_VEL
LIN {X 0,Y 322.095,Z 623.524,A -85,B 0,C 180,E1 -21831.269,E2 -21831.269} C_VEL
LIN {X 0,Y 328.665,Z 629.317,A -85,B 0,C 180,E1 -21834.126,E2 -21834.126} C_VEL
LIN {X 0,Y 333.557,Z 633.261,A -85,B 0,C 180,E1 -21836.349,E2 -21836.349} C_VEL
LIN {X 0,Y 338.202,Z 637.275,A -85,B 0,C 180,E1 -21838.588,E2 -21838.588} C_VEL
LIN {X 0,Y 341.924,Z 640.238,A -85,B 0,C 180,E1 -21840.443,E2 -21840.443} C_VEL
LIN {X 0,Y 346.578,Z 644.394,A -85,B 0,C 180,E1 -21842.96,E2 -21842.96} C_VEL
LIN {X 0,Y 351.284,Z 647.767,A -85,B 0,C 180,E1 -21845.664,E2 -21845.664} C_VEL
LIN {X 0,Y 354.886,Z 651.042,A -85,B 0,C 180,E1 -21847.992,E2 -21847.992} C_VEL
LIN {X 0,Y 358.577,Z 653.635,A -85,B 0,C 180,E1 -21850.538,E2 -21850.538} C_VEL
LIN {X 0,Y 361.105,Z 655.26,A -85,B 0,C 180,E1 -21852.487,E2 -21852.487} C_VEL
LIN {X 0,Y 363.874,Z 657.987,A -85,B 0,C 180,E1 -21854.952,E2 -21854.952} C_VEL
LIN {X 0,Y 366.256,Z 659.916,A -85,B 0,C 180,E1 -21857.441,E2 -21857.441} C_VEL
LIN {X 0,Y 368.08,Z 660.988,A -85,B 0,C 180,E1 -21859.595,E2 -21859.595} C_VEL
LIN {X 0,Y 369.894,Z 661.812,A -85,B 0,C 180,E1 -21862.357,E2 -21862.357} C_VEL
LIN {X 0,Y 371.178,Z 662.568,A -85,B 0,C 180,E1 -21865.107,E2 -21865.107} C_VEL
LIN {X 0,Y 371.897,Z 662.801,A -85,B 0,C 180,E1 -21867.834,E2 -21867.834} C_VEL
LIN {X 0,Y 372.093,Z 662.939,A -85,B 0,C 180,E1 -21870,E2 -21870} C_VEL
LIN {X 0,Y 371.897,Z 662.8,A -85,B 0,C 180,E1 -21872.166,E2 -21872.166} C_VEL
LIN {X 0,Y 371.178,Z 662.573,A -85,B 0,C 180,E1 -21874.892,E2 -21874.892} C_VEL
LIN {X 0,Y 369.894,Z 661.813,A -85,B 0,C 180,E1 -21877.643,E2 -21877.643} C_VEL
LIN {X 0,Y 368.175,Z 661.077,A -85,B 0,C 180,E1 -21880.287,E2 -21880.287} C_VEL
LIN {X 0,Y 365.894,Z 659.661,A -85,B 0,C 180,E1 -21882.967,E2 -21882.967} C_VEL
LIN {X 0,Y 363.333,Z 657.527,A -85,B 0,C 180,E1 -21885.538,E2 -21885.538} C_VEL
LIN {X 0,Y 360.309,Z 654.546,A -85,B 0,C 180,E1 -21888.185,E2 -21888.185} C_VEL
LIN {X 0,Y 357.05,Z 652.623,A -85,B 0,C 180,E1 -21890.537,E2 -21890.537} C_VEL
LIN {X 0,Y 353.237,Z 649.688,A -85,B 0,C 180,E1 -21893.09,E2 -21893.09} C_VEL
LIN {X 0,Y 350.099,Z 646.744,A -85,B 0,C 180,E1 -21895.047,E2 -21895.047} C_VEL
LIN {X 0,Y 345.923,Z 643.868,A -85,B 0,C 180,E1 -21897.394,E2 -21897.394} C_VEL
LIN {X 0,Y 341.231,Z 639.569,A -85,B 0,C 180,E1 -21899.91,E2 -21899.91} C_VEL
LIN {X 0,Y 335.677,Z 635.252,A -85,B 0,C 180,E1 -21902.631,E2 -21902.631} C_VEL
LIN {X 0,Y 331.251,Z 631.295,A -85,B 0,C 180,E1 -21904.722,E2 -21904.722} C_VEL
LIN {X 0,Y 325.728,Z 626.765,A -85,B 0,C 180,E1 -21907.166,E2 -21907.166} C_VEL
LIN {X 0,Y 321.051,Z 622.644,A -85,B 0,C 180,E1 -21909.171,E2 -21909.171} C_VEL
LIN {X 0,Y 315.819,Z 617.992,A -85,B 0,C 180,E1 -21911.335,E2 -21911.335} C_VEL
LIN {X 0,Y 309.217,Z 612.29,A -85,B 0,C 180,E1 -21913.911,E2 -21913.911} C_VEL
LIN {X 0,Y 303.576,Z 607.402,A -85,B 0,C 180,E1 -21915.916,E2 -21915.916} C_VEL
LIN {X 0,Y 296.53,Z 601.391,A -85,B 0,C 180,E1 -21918.21,E2 -21918.21} C_VEL
LIN {X 0,Y 288.504,Z 594.749,A -85,B 0,C 180,E1 -21920.611,E2 -21920.611} C_VEL
LIN {X 0,Y 274.93,Z 582.649,A -85,B 0,C 180,E1 -21924.778,E2 -21924.778} C_VEL
LIN {X 0,Y 266.781,Z 573.404,A -85,B 0,C 180,E1 -21927.817,E2 -21927.817} C_VEL
LIN {X 0,Y 261.37,Z 566.046,A -85,B 0,C 180,E1 -21930.169,E2 -21930.169} C_VEL
LIN {X 0,Y 254.097,Z 554.736,A -85,B 0,C 180,E1 -21933.903,E2 -21933.903} C_VEL
LIN {X 0,Y 249.66,Z 548.043,A -85,B 0,C 180,E1 -21936.562,E2 -21936.562} C_VEL
LIN {X 0,Y 246.926,Z 544.077,A -85,B 0,C 180,E1 -21938.394,E2 -21938.394} C_VEL
LIN {X 0,Y 244.409,Z 540.577,A -85,B 0,C 180,E1 -21940.253,E2 -21940.253} C_VEL
LIN {X 0,Y 241.674,Z 536.755,A -85,B 0,C 180,E1 -21942.543,E2 -21942.543} C_VEL
LIN {X 0,Y 238.442,Z 532.398,A -85,B 0,C 180,E1 -21945.772,E2 -21945.772} C_VEL
LIN {X 0,Y 237.75,Z 531.395,A -85,B 0,C 180,E1 -21946.586,E2 -21946.586} C_VEL
LIN {X 0,Y 235.312,Z 528.607,A -85,B 0,C 180,E1 -21949.888,E2 -21949.888} C_VEL
LIN {X 0,Y 234.377,Z 526.349,A -85,B 0,C 180,E1 -21951.768,E2 -21951.768} C_VEL
LIN {X 0,Y 232.299,Z 524.591,A -85,B 0,C 180,E1 -21960,E2 -21960} C_VEL
LIN {X 0,Y 234.447,Z 526.503,A -85,B 0,C 180,E1 -21967.97,E2 -21967.97} C_VEL
LIN {X 0,Y 236.075,Z 529.757,A -85,B 0,C 180,E1 -21970.886,E2 -21970.886} C_VEL
LIN {X 0,Y 238.31,Z 532.092,A -85,B 0,C 180,E1 -21973.647,E2 -21973.647} C_VEL
LIN {X 0,Y 240.745,Z 535.599,A -85,B 0,C 180,E1 -21976.195,E2 -21976.195} C_VEL
LIN {X 0,Y 241.764,Z 536.836,A -85,B 0,C 180,E1 -21977.118,E2 -21977.118} C_VEL
LIN {X 0,Y 244.649,Z 540.817,A -85,B 0,C 180,E1 -21979.509,E2 -21979.509} C_VEL
LIN {X 0,Y 248.485,Z 546.306,A -85,B 0,C 180,E1 -21982.255,E2 -21982.255} C_VEL
LIN {X 0,Y 251.811,Z 551.263,A -85,B 0,C 180,E1 -21984.355,E2 -21984.355} C_VEL
LIN {X 0,Y 254.955,Z 556.278,A -85,B 0,C 180,E1 -21986.171,E2 -21986.171} C_VEL
LIN {X 0,Y 259.116,Z 564.545,A -85,B 0,C 180,E1 -21988.442,E2 -21988.442} C_VEL
LIN {X 0,Y 264.036,Z 574.936,A -85,B 0,C 180,E1 -21990.879,E2 -21990.879} C_VEL
LIN {X 0,Y 268.713,Z 586.204,A -85,B 0,C 180,E1 -21993.037,E2 -21993.037} C_VEL
LIN {X 0,Y 261.454,Z 683.366,A -85,B 0,C 180,E1 -21995.35,E2 -21995.35} C_VEL
LIN {X 0,Y 259.696,Z 697.91,A -85,B 0,C 180,E1 -21995.806,E2 -21995.806} C_VEL
LIN {X 0,Y 257.39,Z 711.209,A -85,B 0,C 180,E1 -21996.344,E2 -21996.344} C_VEL
LIN {X 0,Y 254.65,Z 723.777,A -85,B 0,C 180,E1 -21997.002,E2 -21997.002} C_VEL
LIN {X 0,Y 251.39,Z 736.369,A -85,B 0,C 180,E1 -21997.837,E2 -21997.837} C_VEL
LIN {X 0,Y 247.521,Z 749.238,A -85,B 0,C 180,E1 -21998.901,E2 -21998.901} C_VEL
LIN {X 0,Y 243.438,Z 761.11,A -85,B 0,C 180,E1 -22000.09,E2 -22000.09} C_VEL
LIN {X 0,Y 239.074,Z 772.433,A -85,B 0,C 180,E1 -22001.444,E2 -22001.444} C_VEL
LIN {X 0,Y 234.291,Z 783.56,A -85,B 0,C 180,E1 -22003.016,E2 -22003.016} C_VEL
LIN {X 0,Y 233.812,Z 784.658,A -85,B 0,C 180,E1 -22003.193,E2 -22003.193} C_VEL
LIN {X 0,Y 231.279,Z 789.393,A -85,B 0,C 180,E1 -22003.843,E2 -22003.843} C_VEL
LIN {X 0,Y 219.743,Z 803.906,A -85,B 0,C 180,E1 -22005.645,E2 -22005.645} C_VEL
